// TIA Portal V16 export
// export: Created 2021-08-10T12:25:23.3020932Z, ExportSetting WithDefaults, DisplayName Totally Integrated Automation Portal, DisplayVersion V16 Update 3, DisplayName TIA Portal Version Control Interface, DisplayVersion V16 Update 2, DisplayName TIA Portal Openness, DisplayVersion V16 Update 3, DisplayName STEP 7 Professional, DisplayVersion V16 Update 3, DisplayName STEP 7 Safety, DisplayVersion V16, DisplayName WinCC Professional, DisplayVersion V16 Update 3
FUNCTION "FC61000_DocGenExample" : Void   // FC61000, LAD
TITLE = Documentation - Gen — Example Documentation (full)
{ S7_Optimized_Access := 'TRUE' }
AUTHOR : M_Gledhill
FAMILY : Documentation
NAME : DocGenExample
VERSION : 1.1
// PRACTICAL SERIES AUTOMATION LIBRARY (PAL)   —   COPYRIGHT 2020 – M. GLEDHILL (MIT LICENCE)
//                   ———— ◆ ————
//  FOR DETAILED DOCUMENTATION — SELECT THE BLOCK IN THE PROJECT TREE AND PRESS SHIFT + F1
//  FULL ONLINE DOCUMENTATION IS AVAILABLE AT: https://practicalseries.com/2001-pal/index.html
// stored: AutoNumber false, IsIECCheckEnabled false, SetENOAutomatically false, UDAEnableTagReadback false
   VAR_INPUT
      SYS_SIGNALS : "UT21000_Dy_SysSignals";   // Common system signals — logic and timing signals
   END_VAR
   VAR_TEMP
      revInfo : "UT01000_St_SysRevision";   // Revision information for this block
      licInfo : "UT01001_St_SysLicence";   // Licence information for this block
      wrkReal : Real;   // Working storage (real)
   END_VAR
BEGIN

REGION Network 1: Block description
   // ▀▀▀▀▀▀▀▀▀▀▀▀▀▀▀▀▀▀▀▀▀▀▀▀▀▀▀▀▀▀▀▀▀▀▀▀▀▀▀▀▀▀▀▀
   // 
   // TITLE:    EXAMPLE DOCUMENTATION FOR USE IN COMMENTS
   // 
   // ▄▄▄▄▄▄▄▄▄▄▄▄▄▄▄▄▄▄▄▄▄▄▄▄▄▄▄▄▄▄▄▄▄▄▄▄▄▄▄▄▄▄▄▄
   // 
   // 
   // 
   // This block contains examples of all the typical forms of documentation used within the PAL
   // software. It provides the following:
   // 
   // CONTENTS (BY NETWORK)
   // 
   // NW 1.    Block Contents
   // NW 2.    Current revision and modification history
   // 
   // 
   // EXAMPLES
   // 
   // NW 3.    Example — Block description — Sections 1 to 3
   // NW 4.    Example — Block description — Sections 4 to 11
   // NW 5.    Example — Current revision and modification history
   // NW 6.    Example — Headings, lists and indented text
   // NW 7.    Example — Body text
   // NW 8.    Example — Standard Tables
   // NW 9.    Example — Other tables
   // NW 10.    Example — Equations
   // NW 11.    Example — Figures
   // 
   // 
   // CHARACTER LISTS
   // 
   // NW 12.    Special characters — Hyphens, whitespace and construction lines
   // NW 13.    Special characters — Arrows, box and block characters
   // NW 14.    Special characters — Currency, punctuation and full-width characters
   // NW 15.    Special characters — Greek, indexing characters and Roman numerals
   // NW 16.    Special characters — Mathematical operators (including vulgar fractions)
   // NW 17.    Special characters — Geometrical and ornamental characters
   // NW 18.    Special characters — Common character widths and additional whitespace characters
   // 
   // 
   // SPECIAL NETWORKS
   // 
   // NW 19.    OB1 NETWORK 1 — Project description
   // NW 20.    OB1 NETWORK 2 — Current revision and modification history
   // 
   // TYPICAL NETWORK COMMENTS
   // 
   // NW 21.    Load the system RTC and store in local variable  [typical network comment]
   // NW 22.    ██ STEP 03340 — DECLARATION (RUNNING)    [sequence network comment]
   // NW 23.       STEP 03340 — ACTION (INITIALISE)           [sequence network comment]
   // NW 24.       STEP 03340 — TRANSITION 01                   [sequence network comment]
   // NW 25.   LICENCE AND CONTACT INFORMATION       [final network]
   // 
   //               ━━━   ⬙⬙⬙⬙⬙⬙   ━━━
   // 
   // 
   // 
   // ▄▄▄▄▄▄▄▄▄▄▄▄▄▄▄▄▄▄▄▄▄▄▄▄▄▄▄▄▄▄▄▄▄▄▄▄▄▄▄▄▄▄▄▄
   // 1.     BLOCK TECHNICAL SUMMARY
   // 
   // 
   //  ――――――――――――――――――――――――――――――――――――――――――
   //  NOMENCLATURE & ADDRESSING
   //  ――――――――――――――――――――――――――――――――――――――――――
   //  BLOCK TITLE         Example Documentation for use in Comments
   //  BLOCK FUNCTION GROUP    Documentation
   //  BLOCK ADDRESS       FC 61000
   //  BLOCK SYMBOL        FC61000_DocGenExample
   //  BLOCK USER ID         DocGenExample
   // 
   //  ――――――――――――――――――――――――――――――――――――――――――
   //  BLOCK TYPE & USAGE
   //  ――――――――――――――――――――――――――――――――――――――――――
   //  BLOCK TYPE         Function (FC)
   //  BLOCK NUMBER        61000
   //  LANGUAGE           LAD
   //  OPTIMISED ACCESS     Yes
   //  PAL USAGE TYPE       Standard block
   // 
   //  ――――――――――――――――――――――――――――――――――――――――――
   //  METRICS
   //  ――――――――――――――――――――――――――――――――――――――――――
   //  EXECUTION TIME       24.48 μs¹
   //  LOAD MEMORY       51.63 kB  (52873 bytes)
   //  WORK MEMORY           0.37 kB      (376 bytes)
   //  ――――――――――――――――――――――――――――――――――――――――――
   //                ¹ Measured on: CPU-1515-2PN (order no. 6ES7 512-2AM02-0AB0)
   // 
   //                ━━━   ⬙⬙⬙⬙⬙⬙   ━━━
   // 
   // 
   // 
   // ▄▄▄▄▄▄▄▄▄▄▄▄▄▄▄▄▄▄▄▄▄▄▄▄▄▄▄▄▄▄▄▄▄▄▄▄▄▄▄▄▄▄▄▄
   // 2.     FUNCTIONAL DESCRIPTION
   // 
   // 
   // FC61000 is a documentation module that contains examples of all the common block and 
   // network comments used throughout the PAL software.
   // 
   // All examples are based upon the Style Guide (Doc. No. PS2001-5-2313-011).
   // 
   // FC61000 also contains lists of the characters available within the Siemens TIA font used within
   // all comment sections.
   // 
   //                ━━━   ⬙⬙⬙⬙⬙⬙   ━━━
   // 
   // 
   // 
   // ▄▄▄▄▄▄▄▄▄▄▄▄▄▄▄▄▄▄▄▄▄▄▄▄▄▄▄▄▄▄▄▄▄▄▄▄▄▄▄▄▄▄▄▄
   // 3.     DETAILED BLOCK DESCRIPTION
   // 
   // 
   // The purpose of this block is to provide an easy point of reference for the various documentation 
   // constructs and styles used within the PAL.
   // 
   // The block itself does not contain any executable code, with the exception of the revision and
   // licence networks, all networks are empty. The block itself does nothing, and its execution will
   // have no effect, other than extending the cycle time.
   // 
   //                ━━━   ⬙⬙⬙⬙⬙⬙   ━━━
   // 
   // 
   // 
   // ▄▄▄▄▄▄▄▄▄▄▄▄▄▄▄▄▄▄▄▄▄▄▄▄▄▄▄▄▄▄▄▄▄▄▄▄▄▄▄▄▄▄▄▄
   // 4.     PARAMETERS
   // 
   // 
   // This block has no parameters.
   // 
   //                ━━━   ⬙⬙⬙⬙⬙⬙   ━━━
   // 
   // 
   // 
   // ▄▄▄▄▄▄▄▄▄▄▄▄▄▄▄▄▄▄▄▄▄▄▄▄▄▄▄▄▄▄▄▄▄▄▄▄▄▄▄▄▄▄▄▄
   // 5.     DATA STRUCTURES AND USAGE (AND INSTANCE DATA BLOCKS)
   // 
   // 
   // The block has the following associated data structure:
   // 
   // 
   //  ――――――――――――――――――――――――――――――――――――――――――
   //  DATA STRUCTURE             DESCRIPTION
   //  ――――――――――――――――――――――――――――――――――――――――――
   //  UT01000_St_SysRevision          Revision information for this block    See FC01001
   //  UT01001_St_SysLicence           Licence information for this block  See FC01001
   //  ――――――――――――――――――――――――――――――――――――――――――
   // 
   // 
   //                ━━━   ⬙⬙⬙⬙⬙⬙   ━━━
   // 
   // 
   // 
   // ▄▄▄▄▄▄▄▄▄▄▄▄▄▄▄▄▄▄▄▄▄▄▄▄▄▄▄▄▄▄▄▄▄▄▄▄▄▄▄▄▄▄▄▄
   // 6.     CONSTANTS AND TEMPORARY (LOCAL) DATA
   // 
   // 
   // The following constants and temporary data storage are used:
   // 
   // 
   //  Temporary (local) data
   //  ――――――――――――――――――――――――――――――――――――――――――
   //  SIGNAL NAME          FUNCTION                  TYPE
   //  ――――――――――――――――――――――――――――――――――――――――――
   //  revInfo             Revision information for the block         UT01000
   //  licInfo           Licensing information for the block      UT01001
   //  wrkReal           Working storage (Real)             Real
   //  ――――――――――――――――――――――――――――――――――――――――――
   // 
   // 
   //  Constants data
   //  ――――――――――――――――――――――――――――――――――――――――――
   //  SIGNAL NAME          FUNCTION                  TYPE
   //  ――――――――――――――――――――――――――――――――――――――――――
   //  _FALSE            Temporary internal "False" signal      Bool
   //  ――――――――――――――――――――――――――――――――――――――――――
   // 
   // 
   //                ━━━   ⬙⬙⬙⬙⬙⬙   ━━━
   // 
   //  
   // 
   // ▄▄▄▄▄▄▄▄▄▄▄▄▄▄▄▄▄▄▄▄▄▄▄▄▄▄▄▄▄▄▄▄▄▄▄▄▄▄▄▄▄▄▄▄
   // 7.     BLOCK CALLS
   // 
   // 
   // There are no PAL block calls from within this block.
   // 
   //                ━━━   ⬙⬙⬙⬙⬙⬙   ━━━
   // 
   // 
   // 
   // ▄▄▄▄▄▄▄▄▄▄▄▄▄▄▄▄▄▄▄▄▄▄▄▄▄▄▄▄▄▄▄▄▄▄▄▄▄▄▄▄▄▄▄▄
   // 8.     ASSOCIATED BLOCKS
   // 
   // 
   // This is a stand-alone block and is not associated with any other blocks.
   // 
   //                ━━━   ⬙⬙⬙⬙⬙⬙   ━━━
   // 
   // 
   // 
   // 9.     SYSTEM BLOCK CALLS AND SYSTEM DATA TYPES
   // 
   // There are no system block calls.
   // 
   //                ━━━   ⬙⬙⬙⬙⬙⬙   ━━━
   // 
   // 
   // 
   // ▄▄▄▄▄▄▄▄▄▄▄▄▄▄▄▄▄▄▄▄▄▄▄▄▄▄▄▄▄▄▄▄▄▄▄▄▄▄▄▄▄▄▄▄
   // 10.     SPECIAL PROPERTIES AND REQUIREMENTS
   // 
   // 
   // 
   // ▂▂▂▂▂▂▂▂▂▂▂▂▂▂▂▂▂▂▂▂▂▂▂▂▂▂▂▂▂▂▂▂▂▂▂▂▂▂▂▂▂▂▂▂
   // 10.1   Block optimisation
   // 
   // 
   // Block optimisation is ACTIVE for this block
   // 
   // 
   // 
   // ▂▂▂▂▂▂▂▂▂▂▂▂▂▂▂▂▂▂▂▂▂▂▂▂▂▂▂▂▂▂▂▂▂▂▂▂▂▂▂▂▂▂▂▂
   // 10.2   Calling requirements
   // 
   // 
   // There are no special calling requirements for this block.
   // 
   //                ━━━   ⬙⬙⬙⬙⬙⬙   ━━━
   // 
   // 
   // 
   // ▄▄▄▄▄▄▄▄▄▄▄▄▄▄▄▄▄▄▄▄▄▄▄▄▄▄▄▄▄▄▄▄▄▄▄▄▄▄▄▄▄▄▄▄
   // 11.     EXAMPLE USAGE
   // 
   // 
   // The following shows a typical deployment of FC61000:
   // 
   // 
   //                        ┌────────────
   //    ────────────────────┤ FC61000 
   //                        ├──────────
   //      "DB21001_DY_StdGlobalData".SysSignals ─┤ SYS_SIGNALS
   //                        │
   //                        │               │
   //                        │               │
   //                                     │
   //                        ─────────────┘
   // 
   //               ━━━   ⬙⬙⬙⬙⬙⬙   ━━━
   // 
   // 
   // ██████████████ █ █ █ █  END   █ █ █ █ ██████████████
END_REGION

REGION Network 2: Current revision and modification history
   // ▄▄▄▄▄▄▄▄▄▄▄▄▄▄▄▄▄▄▄▄▄▄▄▄▄▄▄▄▄▄▄▄▄▄▄▄▄▄▄▄▄▄▄▄
   // MODIFICATION HISTORY
   // 
   // The revision data shown here, in the network comments, contains additional information 
   // reflecting the software development workflow under the version control system (VCS) employed 
   // to track all software changes.
   // 
   // The VCS in use is the Git Source Code Management system in conjunction with the GitHub online 
   // hosting system. The software in its entirety is available in the GitHub remote repository:
   // 
   //      https://github.com/practicalseries/PS2001-pal-software
   // 
   // The repository is public and can be freely copied (forked in GitHub terminology) and used 
   // under the MIT licence. 
   // 
   // The MIT licence is reproduced in full in the last network of this software module.
   // 
   // 
   //  ―――――――――――――――――――――――――――――――――――――――――――
   //  DATE       REVISION             MASTER BRANCH     DEV
   //          (nnn.amm)   COMMIT TAG    (Base ---> Merge)    BRANCH   Author
   //  ———————————————————————————————————————————
   //  2021.08.10    001.102   D0008A-000.103   D0008 N/A     D0008A   M. Gledhill
   //                        Constants table added to network 8
   // 
   //  2021.05.18    001.101   D0005A-000.102   D0005 N/A     D0005A   M. Gledhill
   //                        OB1 secondary commit revision added
   //                        OB1 document list updated
   // 
   //  2021.02.18    001.000   D0002      D0001 D0002  None    M. Gledhill
   //                        FC61000 — RELEASED FOR USE
   //                          Block imported form 000.125-Db
   //  ———————————————————————————————————————————
   //   Where: nnn  =  Major revision
   //         a  =  Type (1-7 Development, 8 Proving, 9 Qualification, 0 Release)
   //       mm  =  Minor revision (must be 00 if a = 0)
   //         Block properties version number should be set to nn.a (only one decimal place)
   // 
   // ▄▄▄▄▄▄▄▄▄▄▄▄▄▄▄▄▄▄▄▄▄▄▄▄▄▄▄▄▄▄▄▄▄▄▄▄▄▄▄▄▄▄▄▄
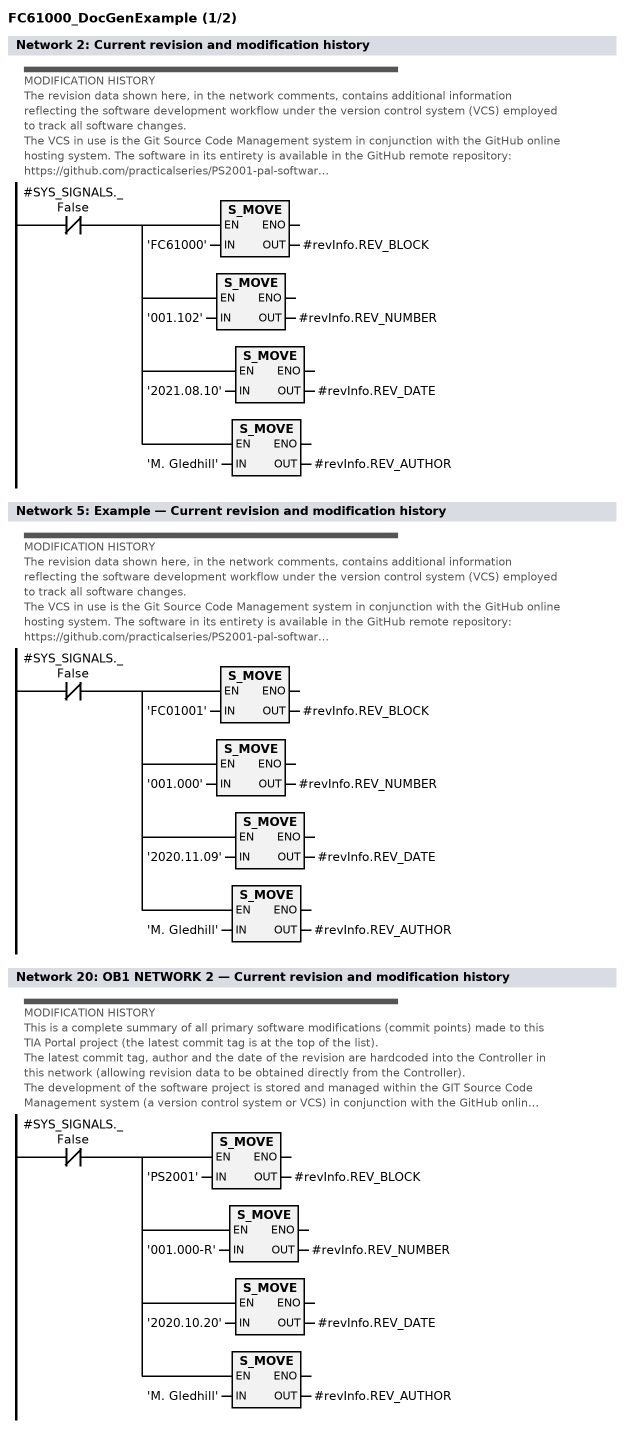
   RUNG wire#powerrail
      I_Contact( #SYS_SIGNALS._False )
      wire#w1
      S_Move(in := 'FC61000', out => #revInfo.REV_BLOCK)
   END_RUNG
   RUNG wire#w1
      S_Move(in := '001.102', out => #revInfo.REV_NUMBER)
   END_RUNG
   RUNG wire#w1
      S_Move(in := '2021.08.10', out => #revInfo.REV_DATE)
   END_RUNG
   RUNG wire#w1
      S_Move(in := 'M. Gledhill', out => #revInfo.REV_AUTHOR)
   END_RUNG
   // the same network as SCL:
   IF NOT #SYS_SIGNALS._False THEN
       #revInfo.REV_BLOCK := 'FC61000';
       #revInfo.REV_NUMBER := '001.102';
       #revInfo.REV_DATE := '2021.08.10';
       #revInfo.REV_AUTHOR := 'M. Gledhill';
   END_IF;
END_REGION

REGION Network 3: Example — Block description — Sections 1 to 3
   // | ▀▀▀▀▀▀▀▀▀▀▀▀▀▀▀▀▀▀▀▀▀▀▀▀▀▀▀▀▀▀▀▀▀▀▀▀▀▀▀▀▀▀▀▀
   // 
   // TITLE:    SUBROUTINE — EVENT TIMER USING RTC
   // 
   // ▄▄▄▄▄▄▄▄▄▄▄▄▄▄▄▄▄▄▄▄▄▄▄▄▄▄▄▄▄▄▄▄▄▄▄▄▄▄▄▄▄▄▄▄
   //  
   // 
   // 
   // This block (FC18151_SubTimeEventRTC) is a subroutine block that times the duration of an event 
   // to nanosecond resolution.
   // 
   // The block records the time the event started (rising edge of the TRIGGER signal), the time the 
   // event ended (falling edge of the TRIGGER signal) and calculates the duration of the event (end 
   // time minus the start time).
   // 
   // The start and end times are read from the real time clock of the controller.
   // 
   // This is a subroutine block.
   // 
   //                ━━━   ⬙⬙⬙⬙⬙⬙   ━━━
   // 
   // 
   // 
   // ▄▄▄▄▄▄▄▄▄▄▄▄▄▄▄▄▄▄▄▄▄▄▄▄▄▄▄▄▄▄▄▄▄▄▄▄▄▄▄▄▄▄▄▄
   // 1.     BLOCK TECHNICAL SUMMARY
   // 
   // 
   //  ――――――――――――――――――――――――――――――――――――――――――
   //  NOMENCLATURE & ADDRESSING
   //  ――――――――――――――――――――――――――――――――――――――――――
   //  BLOCK TITLE         Subroutine Event Timer using RTC
   //  BLOCK FUNCTION GROUP    Subroutine
   //  BLOCK ADDRESS       FC18151
   //  BLOCK SYMBOL        FC18151_SubTimeEventRTC
   //  BLOCK USER ID         SubTimeEventRTC
   // 
   //  ――――――――――――――――――――――――――――――――――――――――――
   //  BLOCK TYPE & USAGE
   //  ――――――――――――――――――――――――――――――――――――――――――
   //  BLOCK TYPE         Function (FC)
   //  BLOCK NUMBER        18151
   //  LANGUAGE           LAD
   //  OPTIMISED ACCESS     Yes
   //  PAL USAGE TYPE       Standard block
   // 
   //  ――――――――――――――――――――――――――――――――――――――――――
   //  METRICS
   //  ――――――――――――――――――――――――――――――――――――――――――
   //  EXECUTION TIME       18.41 μs¹
   //  LOAD MEMORY       23.11 kB  (23667 bytes)
   //  WORK MEMORY           0.43 kB      (442 bytes)
   //  ――――――――――――――――――――――――――――――――――――――――――
   //                ¹ Measured on: CPU-1515-2PN (order no. 6ES7 512-2AM02-0AB0)
   // 
   //                ━━━   ⬙⬙⬙⬙⬙⬙   ━━━
   // 
   // 
   // 
   // ▄▄▄▄▄▄▄▄▄▄▄▄▄▄▄▄▄▄▄▄▄▄▄▄▄▄▄▄▄▄▄▄▄▄▄▄▄▄▄▄▄▄▄▄
   // 2.     FUNCTIONAL DESCRIPTION
   // 
   // 
   // FC18151 is the Subroutine Event Timer using RTC block, it simply records the duration of an event 
   // with a high degree of accuracy. The event being timed is a Boolean signal passed to the block as 
   // the TRIGGER parameter.
   // 
   // Three times are recorded for the event, the start time (rising edge of the TRIGGER parameter), the 
   // end time (falling edge of the TRIGGER parameter) and the duration of the event (end time minus 
   // the start time). The duration is calculated on the falling edge of the TRIGGER parameter, 
   // immediately after the end time is recorded.
   // 
   // The start and end times are read from the Controller’s internal real time clock (RTC) and are 
   // stored in DTL (date time long) format, this format contains year, month, day, hours, minutes, 
   // seconds, milliseconds, microseconds and nano seconds.
   // 
   // The duration is stored in LTime (long time, 64-bit) format, and is very accurate, it resolves to 
   // days, hours, minutes, seconds milliseconds, microseconds and nanoseconds, it keeps this 
   // resolution irrespective of the duration.
   // 
   // The duration is also calculated as a real number in seconds (or fractions thereof); this is a 
   // more convenient format for holding the duration, but is not as accurate as the LTime format.
   // 
   //                ━━━   ⬙⬙⬙⬙⬙⬙   ━━━
   // 
   // 
   // 
   // ▄▄▄▄▄▄▄▄▄▄▄▄▄▄▄▄▄▄▄▄▄▄▄▄▄▄▄▄▄▄▄▄▄▄▄▄▄▄▄▄▄▄▄▄
   // 3.     DETAILED BLOCK DESCRIPTION
   // 
   // 
   // The purpose of this block is to determine with a high degree of accuracy the duration of an event, 
   // the event itself must be in the form of a Boolean trigger signal, the rising edge of the signal is 
   // considered to be the start of the event and the falling edge the end of the event.
   // 
   // The event signal is passed to the block as the TRIGGER parameter. 
   // The block returns five values, these are stored in a UDT passed to the block in the 
   // DYNAMIC_DATA parameter: 
   // 
   // 
   //  ――――――――――――――――――――――――――――――――――――――――――
   //  PARAM         ASSOCIATED UDT            ASSOCIATED DATA BLOCK
   //  ――――――――――――――――――――――――――――――――――――――――――
   //  DYNAMIC_DATA     UT38151_Dy_SubTimeEventRTC       DB38151_Dy_SubTimeEventRTC
   //  ――――――――――――――――――――――――――――――――――――――――――
   // 
   // 
   // The block returns the following data:
   // 
   // 
   //  UT38151_Dy_SubTimeEventRTC
   //  ―――――――――――――――――――――――――――――――――――――――――― 
   //  SIGNAL NAME          FUNCTION                     TYPE
   //  ――――――――――――――――――――――――――――――――――――――――――
   //  status_Running      STATUS — The event timer is running         Bool
   // 
   //  actual_StartTime      ACTUAL — Time at which the TRIGGER signal        DTL
   //                      went high (event start time)
   // 
   //  actual_EndTime        ACTUAL — Time at which the TRIGGER signal     DTL
   //                      went low (event end time)
   // 
   //  actual_Duration        ACTUAL — Event duration              LTime
   // 
   //  actual_DurationSec       ACTUAL — Event duration in seconds           REAL
   //  ――――――――――――――――――――――――――――――――――――――――――
   //  Block returned signals.
   // 
   // 
   // 
   // ▂▂▂▂▂▂▂▂▂▂▂▂▂▂▂▂▂▂▂▂▂▂▂▂▂▂▂▂▂▂▂▂▂▂▂▂▂▂▂▂▂▂▂▂
   // 3.1     Timing an event
   // 
   // 
   // The block constantly monitors the TRIGGER parameter; if a rising edge is seen on the TRIGGER 
   // parameter (point ① in the figure below), the Controller RTC is read and its value is stored in 
   // actual_StartTime, at the same time the running signal (status_Running) is activated.
   // 
   // The block continues to monitor the TRIGGER parameter, when a falling edge is detected 
   // (point ②), the RTC is read once more and its value is stored in actual_EndTime, and the running 
   // signal (status_Running) is deactivated.
   // 
   // Once the end time is stored, the following calculation is carried out:
   // 
   // 
   // ┌───────────────────────────┐
   // │ actual_Duration =  actual_EndTime ─ actual_StartTime    │
   // └───────────────────────────┘
   // 
   // 
   //                     ①            ②
   //   TRIGGER │             ┏━━━━━━━━━━━━┓
   //         │             ┃               ┃
   //         │             ┃               ┃
   //         │             ┃               ┃
   //         │             ┃               ┃                              
   //         ┼━━━━━━━━━━━━╶╶╶╶╶╶╶╶╶╶╶╶╶━━━━━━━━━━ time
   //                  ↗             ↖
   //            actual_StartTime ╎            ╎ actual_EndTime
   //    DTL#2020-04-18-09:34:25.899548353        DTL#2020-04-18-09:34:36.004744916
   // 
   //                    ╎               ╎                      actual_Duration
   //                                      LT#10S_105MS_196US_563NS
   //                    ╎               ╎  
   //                                                     actual_DurationSec
   //                    ╎               ╎                              10.10519
   // 
   //         │status_Running      ┏━━━━━━━━━━━━┓
   //         │             ┃               ┃
   //         │             ┃               ┃
   //         │             ┃               ┃
   //         │             ┃               ┃
   //         ┼━━━━━━━━━━━━╶╶╶╶╶╶╶╶╶╶╶╶╶━━━━━━━━━━
   // 
   // 
   // 
   // ▂▂▂▂▂▂▂▂▂▂▂▂▂▂▂▂▂▂▂▂▂▂▂▂▂▂▂▂▂▂▂▂▂▂▂▂▂▂▂▂▂▂▂▂
   // 3.1     Date and time data types
   // 
   // 
   // Both the start and end times (actual_StartTime and actual_EndTime) are of the type DTL 
   // (date time long), this itself is a data structure in the form:
   // 
   // 
   //  DTL Data Structure
   //  ――――――――――――――――――――――――――――――――――――――――――
   //  SIGNAL NAME          FUNCTION                     TYPE
   //  ――――――――――――――――――――――――――――――――――――――――――
   //  YEAR             Year (returns a value in the range 1970 to 2262)     UInt
   //  MONTH            Month (1-12 representing Jan to Dec)        USInt
   //  DAY              Day of month (1-31)                USInt
   //  WEEKDAY          Day of week (1-7, where 1=Sunday, 7=Saturday)    USInt
   //  HOUR           Hour of day (0-23)                   USInt
   //  MINUTE           Minutes (0-59)                   USInt
   //  SECOND            Seconds (0-59)                  USInt
   //  NANOSECOND        Nanoseconds (0-999,999,999)           UDint
   //  ――――――――――――――――――――――――――――――――――――――――――
   // 
   // 
   // When displayed, it has the format:
   // 
   //       DTL#2020-04-18-09:34:25.899548353
   // 
   //  I.e.      18th April 2020 at 09:43:25 AM and 899,548,353 ns.
   // 
   // The calculated duration (actual_Duration) is of data type LTime (long time).
   // 
   // The LTime data type is essentially an 8-byte number (64-bit number) that stores a time value in 
   // nanoseconds. In the above example, the actual_Duration has the formatted value of:
   // 
   //       LT#10S_105MS_196US_563NS
   // 
   //  I.e.      10 seconds, 105 milliseconds, 196 microseconds and 563 nanoseconds.
   // 
   // It is shown in this format, because TIA portal understands the LTime data type and is able to 
   // interpret the value as days, hours, minute, seconds, milliseconds, microseconds and 
   // nanoseconds. 
   // 
   // In practice, the actual_Duration simply (in this example) holds a very large number:
   // 
   //       10,105,196,563
   // 
   // This is the duration of the event in nanoseconds (i.e. 10,105,196,563 nanoseconds). To convert 
   // the number to seconds, simply divide by 1,000,000,000 (or 1 × 10^9); this would give:
   // 
   //       10.105196563 seconds
   // 
   // The reason the duration is specified as an LTime rather that DTL is that, somewhat confusingly, 
   // DTL is a relative measure of time (relative to 1st January, 1970), if the above duration were 
   // represented as a DTL value it would read:
   // 
   //       DTL#1970-01-01-00:00:10.105196563
   // 
   // Hours, minutes and seconds are OK, but the date part doesn’t make sense (to make it 
   // meaningful, 1970 must be subtracted from the YEAR value and 1 from both the MONTH and 
   // DAY values).
   // 
   // The LTime data type can store a duration of up to 106,751 days (about 300 years) and while not 
   // perfect, it seems long enough for most practical situations (possibly not for geological 
   // applications).
   // 
   // The actual_Duration in LTime format is very accurate, but it is an unwieldly data type, to provide a 
   // more user friendly (although less accurate) format, the actual_Duration signal is converted to a 
   // real number giving the duration in seconds, this is stored in the actual_DurationSec signal. In the 
   // above example: 
   // 
   //       actual_DurationSec has the value 10.10519 seconds
   // 
   // It is less accurate, it does not resolve to nanoseconds; however, it is easier to use and display 
   // and is accurate enough for most applications.
   // 
   // 
   // 
   // ▁▁▁▁▁▁▁▁▁▁▁▁▁▁▁▁▁▁▁▁▁▁▁▁▁▁▁▁▁▁▁▁▁▁▁▁▁▁▁▁▁▁▁▁
   // A note on real numbers
   // 
   // 
   // The LTime format is very accurate, it is basically counting nanoseconds, and because it is 64-bits 
   // long it can count up to very high values (about 584 years at nanosecond resolution).
   // 
   // Real numbers however, are limited to 32-bits and suffer from precision loss, this results from the 
   // fact that the real number has an accuracy of “about” 7 decimal digits, for example 20365.45, 
   // 20.43728, 1.482967, 0.3356428, &c. Essentially, the bigger the number, the fewer the decimal 
   // places — a total of 7 decimal digits.
   // 
   // Very big and very small numbers can be represented by adding trailing zeros for big numbers 
   // (e.g. 3275625000) and leading zeros for small numbers (0.000003275625) in both these 
   // examples, there are only 7 decimal digits, just shifted effectively left or right.
   // 
   // This type of representation is usually handled by applying scientific notation, the number 
   // 1,568,497,000,000 would be represented as 1.568497 × 10^12, it only has 7 decimal digits, 
   // the number 1,568,497,132,792, would be represented as exactly the same value, the 132,792 
   // part of the number cannot be resolved and are lost.
   // 
   //                ━━━   ⬙⬙⬙⬙⬙⬙   ━━━
END_REGION

REGION Network 4: Example — Block description — Sections 4 to 11
   // ▄▄▄▄▄▄▄▄▄▄▄▄▄▄▄▄▄▄▄▄▄▄▄▄▄▄▄▄▄▄▄▄▄▄▄▄▄▄▄▄▄▄▄▄
   // 4.     PARAMETERS
   // 
   // 
   // The following parameters are associated with the block:
   // 
   //  
   //  ――――――――――――――――――――――――――――――――――――――――――
   //  PARAM         FUNCTION                    TYPE      IN-OUT 
   //  ――――――――――――――――――――――――――――――――――――――――――
   //  SYS_SIGNALS      Common system signals              UT21000    In
   //           logic and timing signals for parametric access
   // 
   //  TRIGGER       Event trigger signal (a rising edge marks the     Bool   In
   //           start of the event, the falling edge the end)
   // 
   //  STATIC_DATA     Data structure that holds the configuration data     UT02001    In
   // 
   //  DYNAMIC_DATA      Stores the results of the event timing       UT38151    InOut
   //  ――――――――――――――――――――――――――――――――――――――――――
   // 
   // 
   //                ━━━   ⬙⬙⬙⬙⬙⬙   ━━━
   // 
   // 
   // 
   // ▄▄▄▄▄▄▄▄▄▄▄▄▄▄▄▄▄▄▄▄▄▄▄▄▄▄▄▄▄▄▄▄▄▄▄▄▄▄▄▄▄▄▄▄
   // 5.     DATA STRUCTURES AND USAGE (AND INSTANCE DATA BLOCKS)
   // 
   // 
   // The block has the following associated data structure:
   // 
   // 
   //  ――――――――――――――――――――――――――――――――――――――――――
   //  DATA STRUCTURE             DESCRIPTION
   //  ――――――――――――――――――――――――――――――――――――――――――
   //  UT01000_St_SysRevision          Revision information for this block    See FC01001
   //  UT01001_St_SysLicence           Licence information for this block  See FC01001
   //  UT21000_Dy_SysSignals           System signals for logic and timing  See FC01001
   //  UT38151_Dy_SubTimeEventRTC        Dynamic data structure for the event timing block
   //  ――――――――――――――――――――――――――――――――――――――――――
   // 
   // 
   // 
   // ▂▂▂▂▂▂▂▂▂▂▂▂▂▂▂▂▂▂▂▂▂▂▂▂▂▂▂▂▂▂▂▂▂▂▂▂▂▂▂▂▂▂▂▂
   // 5.1     UT38151_Dy_TimeEventRTC
   // 
   // 
   // Stores the timing values for the event:
   // 
   // 
   //  UT38151_Dy_TimeEventRTC
   //  ――――――――――――――――――――――――――――――――――――――――――
   //  SIGNAL NAME          FUNCTION                     TYPE
   //  ――――――――――――――――――――――――――――――――――――――――――
   //  status_Running      STATUS — The event timer is running         Bool
   // 
   //  actual_StartTime      ACTUAL — Time at which the TRIGGER signal        DTL
   //                      went high (event start time)
   // 
   //  actual_EndTime        ACTUAL — Time at which the TRIGGER signal     DTL
   //                      went low (event end time)
   // 
   //  actual_Duration        ACTUAL — Event duration              LTime
   // 
   //  actual_DurationSec       ACTUAL — Event duration in seconds           REAL
   //  ――――――――――――――――――――――――――――――――――――――――――
   // 
   // 
   //                ━━━   ⬙⬙⬙⬙⬙⬙   ━━━
   // 
   // 
   // 
   // ▄▄▄▄▄▄▄▄▄▄▄▄▄▄▄▄▄▄▄▄▄▄▄▄▄▄▄▄▄▄▄▄▄▄▄▄▄▄▄▄▄▄▄▄
   // 6.     CONSTANTS AND TEMPORARY (LOCAL) DATA
   // 
   // 
   // The following constants and temporary data storage are used:
   // 
   // 
   //  Temporary (local) data
   //  ――――――――――――――――――――――――――――――――――――――――――
   //  SIGNAL NAME          FUNCTION                  TYPE
   //  ――――――――――――――――――――――――――――――――――――――――――
   //  revInfo             Revision information for the block         UT01000
   //  licInfo           Licensing information for the block      UT01001
   //  wrkInt           Working storage area (integer)          Int
   //  wrkReal           Working storage (Real)             Real
   //  wrkLInt            Working storage area (long integer)        LInt
   //  ――――――――――――――――――――――――――――――――――――――――――
   // 
   // 
   //                ━━━   ⬙⬙⬙⬙⬙⬙   ━━━
   // 
   // 
   // 
   // ▄▄▄▄▄▄▄▄▄▄▄▄▄▄▄▄▄▄▄▄▄▄▄▄▄▄▄▄▄▄▄▄▄▄▄▄▄▄▄▄▄▄▄▄
   // 7.     BLOCK CALLS
   // 
   // 
   // There are no PAL block calls from within this block.
   // 
   //                ━━━   ⬙⬙⬙⬙⬙⬙   ━━━
   // 
   // 
   // 
   // ▄▄▄▄▄▄▄▄▄▄▄▄▄▄▄▄▄▄▄▄▄▄▄▄▄▄▄▄▄▄▄▄▄▄▄▄▄▄▄▄▄▄▄▄
   // 8.     ASSOCIATED BLOCKS
   // 
   // 
   // This is a stand-alone block and is not associated with any other blocks.
   // 
   //                ━━━   ⬙⬙⬙⬙⬙⬙   ━━━
   // 
   // 
   // 
   // ▄▄▄▄▄▄▄▄▄▄▄▄▄▄▄▄▄▄▄▄▄▄▄▄▄▄▄▄▄▄▄▄▄▄▄▄▄▄▄▄▄▄▄▄
   // 9.     SYSTEM BLOCK CALLS AND SYSTEM DATA TYPES
   // 
   // 
   // The following calls are made to system blocks:
   // 
   // 
   //  System block calls
   //  ――――――――――――――――――――――――――――――――――――――――――
   //  BLOCK          TITLE             DESCRIPTION  
   //  ――――――――――――――――――――――――――――――――――――――――――
   //  RD_LOC_T             Read the local RTC time    Reads the CPU real time clock 
   //  ――――――――――――――――――――――――――――――――――――――――――
   // 
   // 
   // There are no special system data types used.
   // 
   //                ━━━   ⬙⬙⬙⬙⬙⬙   ━━━
   // 
   // 
   // 
   // ▄▄▄▄▄▄▄▄▄▄▄▄▄▄▄▄▄▄▄▄▄▄▄▄▄▄▄▄▄▄▄▄▄▄▄▄▄▄▄▄▄▄▄▄
   // 10.     SPECIAL PROPERTIES AND REQUIREMENTS
   // 
   // 
   // 
   // ▂▂▂▂▂▂▂▂▂▂▂▂▂▂▂▂▂▂▂▂▂▂▂▂▂▂▂▂▂▂▂▂▂▂▂▂▂▂▂▂▂▂▂▂
   // 10.1   Block optimisation
   // 
   // 
   // Block optimisation is ACTIVE for this block
   // 
   // 
   // 
   // ▂▂▂▂▂▂▂▂▂▂▂▂▂▂▂▂▂▂▂▂▂▂▂▂▂▂▂▂▂▂▂▂▂▂▂▂▂▂▂▂▂▂▂▂
   // 10.2   Calling requirements
   // 
   // 
   // There are no special calling requirements for this block.
   // 
   // 
   // 
   // ▂▂▂▂▂▂▂▂▂▂▂▂▂▂▂▂▂▂▂▂▂▂▂▂▂▂▂▂▂▂▂▂▂▂▂▂▂▂▂▂▂▂▂▂
   // 10.3   Other properties
   // 
   // 
   // This block does not require the usual SYS_SIGNALS logic and timing data.
   // 
   //                ━━━   ⬙⬙⬙⬙⬙⬙   ━━━
   // 
   // 
   // 
   // ▄▄▄▄▄▄▄▄▄▄▄▄▄▄▄▄▄▄▄▄▄▄▄▄▄▄▄▄▄▄▄▄▄▄▄▄▄▄▄▄▄▄▄▄
   // 11.     EXAMPLE USAGE
   // 
   // 
   // The following shows a typical deployment of FC18151:
   // 
   //                      ┌─────────────
   //        ──────────────┤ FC18151
   //                      ├───────────
   //                 %M100.0    │
   //               "Event001"   ─┤ TRIGGER
   //                      │
   //     "DB38151_Dy_TimeEventRTC".Event001 ─┤ DYNAMIC_DATA
   //                      │
   //                      │             │
   //                                    │
   //                           ─────────┘
   // 
   //               ━━━   ⬙⬙⬙⬙⬙⬙   ━━━
   // 
   // 
   // ██████████████ █ █ █ █  END   █ █ █ █ ██████████████
END_REGION

REGION Network 5: Example — Current revision and modification history
   // ▄▄▄▄▄▄▄▄▄▄▄▄▄▄▄▄▄▄▄▄▄▄▄▄▄▄▄▄▄▄▄▄▄▄▄▄▄▄▄▄▄▄▄▄
   // MODIFICATION HISTORY
   // 
   // 
   // The revision data shown here, in the network comments, contains additional information 
   // reflecting the software development workflow under the version control system (VCS) employed 
   // to track all software changes.
   // 
   // The VCS in use is the Git Source Code Management system in conjunction with the GitHub online 
   // hosting system. The software in its entirety is available in the GitHub remote repository:
   // 
   //      https://github.com/practicalseries/PS2001-pal-software
   // 
   // The repository is public and can be freely copied (forked in GitHub terminology) and used 
   // under the MIT licence. 
   // 
   // The MIT licence is reproduced in full in the last network of this software module.
   // 
   // 
   //  ―――――――――――――――――――――――――――――――――――――――――――
   //  DATE       REVISION             MASTER BRANCH     DEV
   //          (nnn.amm)   COMMIT TAG    (Base ---> Merge)    BRANCH   Author
   //  ———————————————————————————————————————————
   //  2020.11.09    001.000   D0003      D0002 D0003  None    M. Gledhill
   //                        FC01001 — RELEASED FOR USE
   //                          Merge back to master branch
   //  
   //  2020.11.09    001.000   D0002A-001.000   D0002 N/A     D0002A   M. Gledhill
   //                        FC01001 — Post test released for use
   // 
   //  2020.11.08    000.801   D0002A-000.801   D0002 N/A     D0002A   M. Gledhill
   //                        FC01001 — Released for SMT
   // 
   //  2020.11.04    000.102   D0002A-000.102   D0002 N/A     D0002A   M. Gledhill
   //                        FC01001 — Incremental build
   // 
   //  2020.11.03    000.101   D0002A-000.101   D0002 N/A     D0002A   M. Gledhill
   //                        FC01001 — Block created
   //  ———————————————————————————————————————————
   //   Where: nnn  =  Major revision
   //         a  =  Type (1-7 Development, 8 Proving, 9 Qualification, 0 Release)
   //       mm  =  Minor revision (must be 00 if a = 0)
   //         Block properties version number should be set to nn.a (only one decimal place)
   // 
   // ▄▄▄▄▄▄▄▄▄▄▄▄▄▄▄▄▄▄▄▄▄▄▄▄▄▄▄▄▄▄▄▄▄▄▄▄▄▄▄▄▄▄▄▄
   RUNG wire#powerrail
      I_Contact( #SYS_SIGNALS._False )
      wire#w1
      S_Move(in := 'FC01001', out => #revInfo.REV_BLOCK)
   END_RUNG
   RUNG wire#w1
      S_Move(in := '001.000', out => #revInfo.REV_NUMBER)
   END_RUNG
   RUNG wire#w1
      S_Move(in := '2020.11.09', out => #revInfo.REV_DATE)
   END_RUNG
   RUNG wire#w1
      S_Move(in := 'M. Gledhill', out => #revInfo.REV_AUTHOR)
   END_RUNG
   // the same network as SCL:
   IF NOT #SYS_SIGNALS._False THEN
       #revInfo.REV_BLOCK := 'FC01001';
       #revInfo.REV_NUMBER := '001.000';
       #revInfo.REV_DATE := '2020.11.09';
       #revInfo.REV_AUTHOR := 'M. Gledhill';
   END_IF;
END_REGION

REGION Network 6: Example — Headings, lists and indented text
   // ▀▀▀▀▀▀▀▀▀▀▀▀▀▀▀▀▀▀▀▀▀▀▀▀▀▀▀▀▀▀▀▀▀▀▀▀▀▀▀▀▀▀▀▀
   // ↳
   // TITLE:    HEADINGS, LISTS AND INDENTED TEXT
   // ↳
   // ▄▄▄▄▄▄▄▄▄▄▄▄▄▄▄▄▄▄▄▄▄▄▄▄▄▄▄▄▄▄▄▄▄▄▄▄▄▄▄▄▄▄▄▄[3 empty lines below]
   // ↳
   // ↳
   // ↳
   // Lorem ipsum dolor sit amet, consectetur adipiscing elit, sed do eiusmod tempor incididunt ut 
   // labore et dolore magna aliqua. Euismod lacinia at quis risus sed. Semper feugiat nibh sed 
   // pulvinar proin gravida hendrerit.
   // ↳
   //                ━━━   ⬙⬙⬙⬙⬙⬙   ━━━[1 empty line above]
   // ↳
   // ↳
   // ↳
   // ▄▄▄▄▄▄▄▄▄▄▄▄▄▄▄▄▄▄▄▄▄▄▄▄▄▄▄▄▄▄▄▄▄▄▄▄▄▄▄▄▄▄▄▄[3 empty lines above, 2 after title]
   // 1.     [MAIN SECTION — ALL UPPERCASE — IF UNNUMBERED STARTS AT LEFT EDGE]
   // 10.     [MAIN SECTION — ALL UPPERCASE — IF UNNUMBERED STARTS AT LEFT EDGE]
   // ↳
   // ↳
   // Lorem ipsum dolor sit amet, consectetur adipiscing elit, sed do eiusmod tempor incididunt ut 
   // labore et dolore magna aliqua. Euismod lacinia at quis risus sed. Semper feugiat nibh sed 
   // pulvinar proin gravida hendrerit.
   // ↳
   //                ━━━   ⬙⬙⬙⬙⬙⬙   ━━━[1 empty line above]
   // ↳
   // ↳
   // ↳
   // ▂▂▂▂▂▂▂▂▂▂▂▂▂▂▂▂▂▂▂▂▂▂▂▂▂▂▂▂▂▂▂▂▂▂▂▂▂▂▂▂▂▂▂▂[3 empty lines above, 2 after title]
   // 1.1     [Subsection, two single digits   — Sentence case — if unnumbered, starts at left edge]
   // 10.1   [Subsection, one double digit   — Sentence case — if unnumbered, starts at left edge]
   // 10.10    [Subsection, two double digits — Sentence case — if unnumbered, starts at left edge]
   // ↳
   // ↳
   // Lorem ipsum dolor sit amet, consectetur adipiscing elit, sed do eiusmod tempor incididunt ut 
   // labore et dolore magna aliqua. Euismod lacinia at quis risus sed. Semper feugiat nibh sed 
   // pulvinar proin gravida hendrerit.
   // ↳
   //                ━━━   ⬙⬙⬙⬙⬙⬙   ━━━[1 empty line above]
   // ↳
   // ↳
   // ↳
   // ▁▁▁▁▁▁▁▁▁▁▁▁▁▁▁▁▁▁▁▁▁▁▁▁▁▁▁▁▁▁▁▁▁▁▁▁▁▁▁▁▁▁▁▁[3 empty lines above, 2 after title]
   // 1.1.1     [Inline, three single digits   — Sentence case — if unnumbered, starts at left edge]
   // 10.1.1   [Inline, one double digit   — Sentence case — if unnumbered, starts at left edge]
   // 10.10.1   [Inline, two double digits    — Sentence case — if unnumbered, starts at left edge]
   // 10.10.10 [Inline, three double digits — Sentence case — if unnumbered, starts at left edge]
   // ↳
   // ↳
   //    •   [Lists — non-numbered]
   //    ① [Lists — numbered]
   //    1.  [Lists — numbered single digit   — less than 10 entries]
   //      1.  [Lists — numbered single digit   — 10 or more entries]
   //    10.  [Lists — numbered double digit — 10 or more entries]
   // 
   //    1.  Communication handling
   //      Executes system to system communications (Controller to Controller, point-to-point,
   //      ProfiBus FMS &c.)
   //    2.  Subroutine functions
   //      Various subroutines (called by other block) to execute particular functions 
   //      (subroutines are organised into similar function areas)
   //    3.  Normal (non-error) interrupt functions
   //      Usually associated with specific OBs, interrupts generated by standard system events
   //      (time of day, cyclic, hardware &c.)
   // 
   // Note:    Bipolar and unipolar instruments have different tolerances, a 0-20 mA unipolar signal
   //      has a full instrument range of 16 mA and the 2.5% tolerance will thus be ±0.4 mA 
   // 
   // ――――――――――
   // ¹         Footnotes can use the characters ¹, ² and ³ to indicate the footnote number
   //      Second lines are identical to those for notes.
   // ――――――――――
   // ↳
   //                ━━━   ⬙⬙⬙⬙⬙⬙   ━━━
   // ↳
   // ↳
   // ██████████████ █ █ █ █  END   █ █ █ █ ██████████████
   // ↳
END_REGION

REGION Network 7: Example — Body text
   // ▀▀▀▀▀▀▀▀▀▀▀▀▀▀▀▀▀▀▀▀▀▀▀▀▀▀▀▀▀▀▀▀▀▀▀▀▀▀▀▀▀▀▀▀
   // 
   // TITLE:    BODY TEXT (AN EXAMPLE)
   // 
   // ▄▄▄▄▄▄▄▄▄▄▄▄▄▄▄▄▄▄▄▄▄▄▄▄▄▄▄▄▄▄▄▄▄▄▄▄▄▄▄▄▄▄▄▄
   // 
   // 
   // Normal (body) text is left justified to the left hand edge of the comment area; manual line-breaks
   // must be inserted when the text exceeds the range of the title bars (lines at the top of this block
   // and above each section and subsection — exactly 44 em-spaces).
   // 
   // The following fragment highlights this: 
   // 
   // The alignments in Figure 7.4 are such that the leading edge (left side) of any indented character
   // is aligned with the leading edge of an em-space in a line of em-spaces that span the page (this
   // can be seen with the chequered patterns in the screen shot — all indents line up with the left
   // edge of an em-space).
   // 
   // The problem with this is that the alphanumeric characters are not all the same width and
   // generally, they are not one em-space wide (there are no characters that are one em wide, not
   // even the M, which is odd given that that is how the em unit was derived, see here).
   // With the TIA Portal font, one em is exactly the same width as four normal space characters (a 
   // normal space being the character entered when the space bar is pressed). The alphanumeric 
   // characters (and in fact, all the characters) in the TIA Portal font have the peculiarity that they are
   // all a multiple of ⅓ of a normal space , the “i" for example is one normal space wide, “a” is 2⅓
   // normal space characters wide and “m” is 2⅔ normal space characters wide.
   // 
   // This “feature?” of the font is a distinct advantage; it means that is possible to always bring things
   // back into true alignment by using the range of whitespace characters. There are five such 
   // whitespace characters.
   // 
   // The width of the page is approximately 3.38 lowercase alphabets:
   // 
   // abcdefghijklmnopqrstuvwxyzabcdefghijklmnopqrstuvwxyzabcdefghijklmnopqrstuvwxyzabcdefghij
   // 
   // This averages at about 78 (non-space) characters per line.
   // 
   // A comment field can contain 65000 characters (approx.) including spaces and line breaks.
   // 
   // This broadly equates to 670 lines of standard text, approximately 13000 words.
   // ↳
   //                ━━━   ⬙⬙⬙⬙⬙⬙   ━━━
   // ↳
   // ↳
   // ██████████████ █ █ █ █  END   █ █ █ █ ██████████████
   // ↳
END_REGION

REGION Network 8: Example — Standard Tables
   // ▀▀▀▀▀▀▀▀▀▀▀▀▀▀▀▀▀▀▀▀▀▀▀▀▀▀▀▀▀▀▀▀▀▀▀▀▀▀▀▀▀▀▀▀
   // 
   // TITLE:    STANDARD TABLES (EXAMPLES)
   // 
   // ▄▄▄▄▄▄▄▄▄▄▄▄▄▄▄▄▄▄▄▄▄▄▄▄▄▄▄▄▄▄▄▄▄▄▄▄▄▄▄▄▄▄▄▄
   // 
   // 
   // 
   // Tables always have 2 blank lines above and 2 blank lines below.
   // 
   // ▌▌▌▌▌▌▌▌▌▌▌▌▌▌▌▌▌▌PARAMETER TABLE▐▐▐▐▐▐▐▐▐▐▐▐▐▐▐▐▐▐
   // ↳
   // ↳
   //  ――――――――――――――――――――――――――――――――――――――――――
   //  PARAM         FUNCTION                    TYPE      IN-OUT 
   //  ――――――――――――――――――――――――――――――――――――――――――
   //  SYS_SIGNALS      The system logic and timing signals for       UT21000    In
   //           parametric access
   // 
   //  RAW_ANALOG      The unscaled analogue input (input word         Word     In
   //           address for the IO card to which the instrument 
   //           is connected)
   // 
   //  RAW_MIN     Minimum value of the analogue input range      Int      In
   //           (see Table 3.1 to Table 3.3 for typical values)
   // 
   //  RAW_MAX       Maximum value of the analogue input range      Int      In
   //           (see Table 3.1 to Table 3.3 for typical values)
   // 
   //  SCALE_MIN    Calibrated lower value of the instrument       Real      In
   //           range in engineering units
   // 
   //  SCALE_MAX      Calibrated upper value of the instrument      Real      In
   //           range in engineering units
   // 
   //  STATIC_DATA     The static data associated with the PID loop       UT10001 In
   // 
   //  DYNAMIC_DATA      Stores the results of the event timing       UT38151    InOut
   //  ――――――――――――――――――――――――――――――――――――――――――
   // ↳
   // ↳
   // 
   // ▌▌▌▌▌▌▌▌▌▌▌▌▌▌▌▌▌ DATA STRUCTURE LIST ▐▐▐▐▐▐▐▐▐▐▐▐▐▐▐▐▐
   // ↳
   // ↳
   //  ――――――――――――――――――――――――――――――――――――――――――
   //  DATA STRUCTURE             DESCRIPTION
   //  ――――――――――――――――――――――――――――――――――――――――――
   //  UT01000_St_SysRevision          Revision information for this block    See FC01000
   //  UT01001_St_SysLicence           Licence information for this block  See FC01000
   //  UT21000_Dy_SysSignals           System signals for logic and timing  See FC01000
   // 
   //  UT02001_St_InstAnalogRead      Static data structure for an analogue instrument.
   //                     Holds configuration information, instrument ranges 
   //                     and scaling, alarm/warning thresholds &c.
   // 
   //  UT22001_Dy_InstAnalogRead        Dynamic data structure for an analogue instrument.
   //                     Current scaled instrument reading, alarm status, 
   //                     operating modes, timer values &c.
   //  ――――――――――――――――――――――――――――――――――――――――――
   // ↳
   // ↳
   // 
   // ▌▌▌▌▌▌▌▌▌▌   DATA STRUCTURE CONTENTS AND INSTANCE DBs   ▐▐▐▐▐▐▐▐▐▐
   // ↳
   // ↳
   //  UT38151_Dy_TimeEventRTC
   //  ――――――――――――――――――――――――――――――――――――――――――
   //  SIGNAL NAME          FUNCTION                     TYPE
   //  ――――――――――――――――――――――――――――――――――――――――――
   //  status_Running      STATUS — The event timer is running         Bool
   // 
   //  actual_StartTime      ACTUAL — Time at which the TRIGGER signal        DTL
   //                      went high (event start time)
   // 
   //  actual_EndTime        ACTUAL — Time at which the TRIGGER signal     DTL
   //                      went low (event end time)
   // 
   //  actual_Duration        ACTUAL — Event duration              LTime
   // 
   //  actual_DurationSec       ACTUAL — Event duration in seconds           REAL
   //  ――――――――――――――――――――――――――――――――――――――――――
   // ↳
   // ↳
   // 
   // ▌▌▌▌▌▌▌▌▌▌▌▌▌▌▌  CONSTANTS AND LOCAL DATA  ▐▐▐▐▐▐▐▐▐▐▐▐▐▐▐
   // 
   // [Keep local and constant data function description to one line and no gaps between rows]
   // ↳
   // ↳
   //  CONSTANTS DATA
   //  ――――――――――――――――――――――――――――――――――――――――――
   //  SIGNAL NAME       Value    FUNCTION                  TYPE
   //  ――――――――――――――――――――――――――――――――――――――――――
   //  k_TIME_OP_MIN      0.21      Minimum value for the operation timer     Real
   //  ――――――――――――――――――――――――――――――――――――――――――
   // ↳
   // ↳
   //  TEMPORARY (LOCAL) DATA
   //  ――――――――――――――――――――――――――――――――――――――――――
   //  SIGNAL NAME          FUNCTION                     TYPE
   //  ――――――――――――――――――――――――――――――――――――――――――
   //  wrkPercentPV          Process Variable as a percentage of inst. range     Real
   //  wrkPercentSP          Setpoint as a percentage of PV instrument range     Real
   //  wrkPercentDB         Deadband as a percentage of PV instrument range    Real
   //  wrkGain          Gain (adjusted for reverse/normal Acting)      Real
   //  wrkCycTime          Cyclic execution time (TIME format)         Time
   //  ――――――――――――――――――――――――――――――――――――――――――
   // ↳
   // ↳
   // 
   // ▌▌▌▌▌▌▌▌▌▌▌▌▌▌▌▌▌▌▌  BLOCK LIST  ▐▐▐▐▐▐▐▐▐▐▐▐▐▐▐▐▐▐▐
   // ↳
   // ↳
   //  BLOCK CALLS
   //  ――――――――――――――――――――――――――――――――――――――――――
   //  BLOCK          TITLE             DESCRIPTION  
   //  ――――――――――――――――――――――――――――――――――――――――――
   //  FC18001         StdSubScaleAI        Scales an analogue input signal 
   //                            Continuation line
   //  ――――――――――――――――――――――――――――――――――――――――――
   // ↳
   // ↳
   //  ASSOCIATED BLOCKS
   //  ――――――――――――――――――――――――――――――――――――――――――
   //  BLOCK          TITLE             DESCRIPTION  
   //  ――――――――――――――――――――――――――――――――――――――――――
   //  FC17102         StdCommsWrite65K       Write data partner block
   //                            Continuation line 
   //  ――――――――――――――――――――――――――――――――――――――――――
   // ↳
   // ↳
   // 
   // ▌▌▌▌▌▌▌▌▌▌▌▌▌▌▌▌▌  SYSTEM BLOCK LIST   ▐▐▐▐▐▐▐▐▐▐▐▐▐▐▐▐▐
   // ↳
   // ↳
   //  SYSTEM BLOCK CALLS
   //  ――――――――――――――――――――――――――――――――――――――――――
   //  BLOCK          TITLE             DESCRIPTION  
   //  ――――――――――――――――――――――――――――――――――――――――――
   //  RD_LOC_T             Read the local RTC time    Reads the CPU real time clock 
   //  (FC804)                        Continuation line 
   //                            Continuation line
   //  ――――――――――――――――――――――――――――――――――――――――――
   // ↳
   // ↳
   // 
   // ▌▌▌▌▌▌▌▌▌▌▌▌▌▌▌▌▌▌▌▌▌▌▐▐▐▐▐▐▐▐▐▐▐▐▐▐▐▐▐▐▐▐▐▐
   // ↳
   //                ━━━   ⬙⬙⬙⬙⬙⬙   ━━━
   // ↳
   // ↳
   // ██████████████ █ █ █ █  END   █ █ █ █ ██████████████
   // ↳
END_REGION

REGION Network 9: Example — Other tables
   // ▀▀▀▀▀▀▀▀▀▀▀▀▀▀▀▀▀▀▀▀▀▀▀▀▀▀▀▀▀▀▀▀▀▀▀▀▀▀▀▀▀▀▀▀
   // 
   // TITLE:    OTHER TABLES (EXAMPLES)
   // 
   // ▄▄▄▄▄▄▄▄▄▄▄▄▄▄▄▄▄▄▄▄▄▄▄▄▄▄▄▄▄▄▄▄▄▄▄▄▄▄▄▄▄▄▄▄
   // 
   // 
   // 
   // Tables always have 2 blank lines above and 2 blank lines below.
   // 
   // 
   // ▌▌▌▌▌▌▌▌▌▌▌▌▌▌▌▌▌  TWO COLUMN TABLE ▐▐▐▐▐▐▐▐▐▐▐▐▐▐▐▐▐
   // ↳
   // ↳
   //  ――――――――――――――――――――――――――――――――――――――――――
   //  IO TYPE            DESCRIPTION
   //  ――――――――――――――――――――――――――――――――――――――――――
   //  ET200MP         Standard IO high density IO for the S7-1500 range
   // 
   //  ET200M           Standard IO high density IO for the S7-300 range, 
   //               can be used as remote IO for the S7-1500
   //  ――――――――――――――――――――――――――――――――――――――――――
   // ↳
   // ↳
   // 
   // ▌▌▌▌▌▌▌▌▌▌▌▌▌▌▌▌▌THREE COLUMN TABLE ▐▐▐▐▐▐▐▐▐▐▐▐▐▐▐▐▐
   // 
   // [Numerical table with number alignment to the right]
   // ↳
   // ↳
   //  ――――――――――――――――――――――――――――――――――――――――――
   //  PRESSURE           RAW SIGNAL           SCALED VAL
   //  ――――――――――――――――――――――――――――――――――――――――――
   //  -250.0 Pa                   0             -250.0 Pa
   //        0.0 Pa                  13824            0.0 Pa
   //   250.0 Pa                  27648              250.0 Pa
   //  ――――――――――――――――――――――――――――――――――――――――――
   // ↳
   // ↳
   // 
   // ▌▌▌▌▌▌▌▌▌▌▌▌▌▌▌▌▌ FOUR COLUMN TABLE ▐▐▐▐▐▐▐▐▐▐▐▐▐▐▐▐▐
   // 
   // [Numerical table with number alignment to the right]
   // ↳
   // ↳
   //  ――――――――――――――――――――――――――――――――――――――――――
   //  RAW MIN       RAW MAX      SCALED MIN       SCALED MAX
   //  ――――――――――――――――――――――――――――――――――――――――――
   //        0        27648        -250.0 Pa        250.0 Pa
   //  ――――――――――――――――――――――――――――――――――――――――――
   // ↳
   // ↳
   // 
   // ▌▌▌▌▌▌▌▌▌▌▌▌▌▌▌▌▌  TABLE WITH HEADING  ▐▐▐▐▐▐▐▐▐▐▐▐▐▐▐▐▐
   // 
   // [Numerical table with number alignment to the right]
   // ↳
   // ↳
   //  CURRENT SIGNALS
   //  ――――――――――――――――――――――――――――――――――――――――――
   //  SIGNAL TYPE     SIG MIN VAL      RAW_MIN     SIG MAX VAL     RAW_MAX
   //  ――――――――――――――――――――――――――――――――――――――――――
   //    4-20 mA      4 mA          0          20 mA       27648
   //    0-20 mA      0 mA          0          20 mA       27648
   //  -20 to 20 mA      -20 mA      -27648          20 mA       27648
   //  ――――――――――――――――――――――――――――――――――――――――――
   // ↳
   // ↳
   // 
   // ▌▌▌▌▌▌▌▌▌▌▌▌▌▌▌▌▌▌▌▌▌▌▐▐▐▐▐▐▐▐▐▐▐▐▐▐▐▐▐▐▐▐▐▐
   // ↳
   //                ━━━   ⬙⬙⬙⬙⬙⬙   ━━━
   // ↳
   // ↳
   // ██████████████ █ █ █ █  END   █ █ █ █ ██████████████
   // ↳
END_REGION

REGION Network 10: Example — Equations
   // ▀▀▀▀▀▀▀▀▀▀▀▀▀▀▀▀▀▀▀▀▀▀▀▀▀▀▀▀▀▀▀▀▀▀▀▀▀▀▀▀▀▀▀▀
   // 
   // TITLE:    EQUATIONS (EXAMPLES)
   // 
   // ▄▄▄▄▄▄▄▄▄▄▄▄▄▄▄▄▄▄▄▄▄▄▄▄▄▄▄▄▄▄▄▄▄▄▄▄▄▄▄▄▄▄▄▄
   // 
   // 
   // 
   // ┌─────────────────────────────────────┐
   // │                                                                                                              100                         │
   // │ SigPercent = (Signal ─ PV_RANGE_MIN) ╳ ---------------------------------------------------------------    │
   // │                    (PV_RANGE_MAX ─ PV_RANGE_MIN)    │
   // └─────────────────────────────────────┘
   // 
   // 
   // ┌───────────────────────┐
   // │        2.5               │
   // │ CalcValOOR = ------------ ╳ (RAW_MAX ─ RAW_MIN)   │
   // │       100               │
   // └───────────────────────┘
   // 
   // Mathematical operators:
   //    Large:  ┼ ─ ╳
   //    Small: + − × ÷ ± ≤ ≥
   // ↳
   //                ━━━   ⬙⬙⬙⬙⬙⬙   ━━━
   // ↳
   // ↳
   // ██████████████ █ █ █ █  END   █ █ █ █ ██████████████
   // ↳
END_REGION

REGION Network 11: Example — Figures
   // ▀▀▀▀▀▀▀▀▀▀▀▀▀▀▀▀▀▀▀▀▀▀▀▀▀▀▀▀▀▀▀▀▀▀▀▀▀▀▀▀▀▀▀▀
   // 
   // TITLE:    FIGURES (EXAMPLES)
   // 
   // ▄▄▄▄▄▄▄▄▄▄▄▄▄▄▄▄▄▄▄▄▄▄▄▄▄▄▄▄▄▄▄▄▄▄▄▄▄▄▄▄▄▄▄▄
   // 
   // 
   // 
   // Some example figures, always pad gaps with an EM-SPACE, where text is used add normal 
   // spaces with either a THREE-PER-EM space or a SIX-PER-EM space — one of these will give an
   // exact alignment.
   // 
   // These figures are included to show what is possible.
   // 
   // 
   // Figures have 1 blank line above and 1 below.
   // 
   //   → ┌────────┐
   // ┌───┤   IDLE   │
   // │   └───┬────┘
   // │       ↓
   // │       START
   // │       │
   // │   ┌───┴────┐ →
   // │   │  STARTING     ├───┐
   // │   └───┬────┘   │
   // │       ↓        │
   // │         Run*       ├────────────────────┐
   // │       │        │                    │
   // │   ┌───┴────┐ → │                    │
   // │   │        ├───┴───  Hold  ───┐          │
   // │   │        │             ↓          ↓
   // │   │        │         ┌───┴────┐ ┌───┴────┐
   // │   │        │         │  HOLDING    │ │ ErrHOLDING   │
   // │   │        │         └───┬────┘ └───┬────┘
   // │   │        │             Held*        ErrHeld*
   // │   │        │         ┌───┴────┐ ┌───┴────┐
   // │   │        │         │   HELD    │ │  ErrHELD   │
   // │   │  RUNNING     │         └───┬────┘ └───┬────┘
   // │   │        │              Resume         ErrResume
   // │   │        │         ┌───┴────┐ ┌───┴────┐
   // │  ┌┤        │         │   RESUMING    │ │  ErrRESUMING   │ 
   // │  ││        │         └───┬────┘ └───┬────┘  
   // │  ││        │             │          │
   // │  ││        │ ←           ↓          ↓
   // │  ││        │─────────────┴──────────┘
   // │  │└───┬────┘   Returns to previous step (running or starting)
   // │  ↓    ↓
   // │  │    │
   // │ Complete Complete*     Note: *indicates that the command is issued
   // │  │    │           automatically by the sequence (it
   // │  │┌───┴────┐      can also be triggered manually):
   // │  └┤ COMPLETING  │          1. Run
   // │   └───┬────┘          2. Complete
   // │       ↓               3. Completed
   // ↑     Completed*              4. Held
   // │       │               5. ErrHeld
   // │   ┌───┴────┐          6. Stopped
   // │   │  COMPLETED   │          7. Aborted
   // │   └───┬────┘
   // │       │
   // │              RetIdle*
   // │   ←   ↓
   // ├───────┘
   // │   
   // │
   // │     ABORT ROUTE                  STOPPING ROUTE
   // │Can be triggered in all states except       Can be triggered in all states except
   // │ IDLE, COMPLETED, ABORTING or            IDLE, COMPLETED, ABORTING, 
   // │       ABORTED                 ABORTED, STOPPING or STOPPED
   // │       │                       │
   // │       ↓                       ↓
   // │                Abort                                                                                       Stop
   // │       │                       │
   // │   ┌───┴────┐              ┌───┴────┐
   // ↑   │ ABORTING    │              │  STOPPING    │
   // │   └───┬────┘              └───┬────┘
   // │       ↓                       ↓
   // │              Aborted*                                                                                Stopped*
   // │       │                       │
   // │   ┌───┴────┐              ┌───┴────┐
   // │   │ ABORTED      │              │ STOPPED   │
   // │   └───┬────┘              └───┬────┘
   // │       │                       │
   // │      RetIdle (*)                                                                               RetIdle (*)
   // │  ←    ↓                       ↓
   // └───────┴───────────────────────┘
   // 
   // 
   // 
   // ▌▌▌▌▌▌▌▌▌▌▌▌▌▌▌▌▌▌   INLINE FIGURES ▐▐▐▐▐▐▐▐▐▐▐▐▐▐▐▐▐▐
   // 
   // 
   // 
   // ▂▂▂▂▂▂▂▂▂▂▂▂▂▂▂▂▂▂▂▂▂▂▂▂▂▂▂▂▂▂▂▂▂▂▂▂▂▂▂▂▂▂▂▂
   // 1.1     Step operation and phases
   // 
   // 
   //  ┌─────┐  The sequence progresses from one step to the next if the
   //  │Step n        │  transition logic for the step is TRUE. 
   //  └┬────┘                                                                 
   //   │       In this example, STEP n is active and will remain active
   //         --- T n        until its associated transition (T n) becomes TRUE; at this
   //   │       point the sequence will advance to the next step (STEP n+1)
   //  ┌┴────┐  and execute the actions required of this step. The sequence
   //  │Step n+1    │  will remain in this step until its transition condition is
   //  └┬────┘  true, at which point the sequence will advance again.
   //   │                                                                      
   //         --- T n+1      Each step has a step number, this is an integer value in
   //   │       the range 0 to 29999; step numbers are assigned in specific
   //           Ranges for different operating states of the sequence (IDLE,
   //           STARTING, RUNNING &c.).
   // 
   // Within an individual step, the step has three distinct phases and actions can 
   // be attached to any of these phases (externally to the block). The phases are:
   // 
   // INITIALISING (Phs_INIT)                   ┌──────┐
   // This is activated for a single OB1 scan when the step   │INITIALISING   │
   // is first processed (I.e. on the rising edge of the step     └┬─────┘
   // becoming active).                     │      
   //                           ┌┴─────┐ 
   // PROCESSING (Phs_PROC)               │PROCESSING │
   // This is the main phase of the step, it is activated        └┬─────┘
   // immediately following the INITIALISING phase and remains  │       
   // active until the step TRANSITION condition is TRUE. The     --- T n   
   // PROCESSING phase becomes inactive on the rising edge   │     
   // of the TRANSITION condition.              ┌┴─────┐
   //                           │TERMINATING │    
   // TERMINATING (Phs_TERM)               └──────┘    
   // The TERMINATING phase is activated on the rising edge of the TRANSITION
   // condition (the same condition that terminates the PROCESSING phase). The
   // terminating phase is active for a single OB1 scan.
   // 
   // 
   // [ALTERNATIVE]
   //  ┌──────┐ INITIALISING (Phs_INIT)
   //  │INITIALISING   │ This is activated for a single OB1 scan when the step
   //  └┬─────┘ is first processed (I.e. on the rising edge of the step
   //   │       becoming active).
   //  ┌┴─────┐    
   //  │PROCESSING │ PROCESSING (Phs_PROC)
   //  └┬─────┘ This is the main phase of the step, it is activated 
   //   │       immediately following the INITIALISING phase and remains
   //          --- T n       active until the step TRANSITION condition is TRUE. The
   //   │       PROCESSING phase becomes inactive on the rising edge
   //  ┌┴─────┐ of the TRANSITION condition.
   //  │TERMINATING │    
   //  └──────┘
   // 
   // TERMINATING (Phs_TERM)
   // The TERMINATING phase is activated on the rising edge of the TRANSITION
   // condition (the same condition that terminates the PROCESSING phase). The
   // terminating phase is active for a single OB1 scan.
   // 
   // 
   // 
   // 
   // ▌▌▌▌▌▌▌▌▌▌▌▌▌▌▌▌▌   GRAPHICAL FIGURE   ▐▐▐▐▐▐▐▐▐▐▐▐▐▐▐▐▐
   // 
   //     No. of scans from start of STEP 1
   //     1      2      3     4      5     6       7      8      9
   //   ┼─┼─┼─┼─┼─┼─┼─┼─┼─┼─┼─┼  ─ ─ ┐
   //                                │
   //   ┌─┐                          │
   //   │ │               Phs_INIT
   //  ─┘ └────────────────────                   
   //   ┼─┼─┼─┼─┼─┼─┼─┼─┼─┼─┼─┼                   
   //  
   //     ┌───┐                       S
   //     │   │           Phs_PROC      T
   //  ───┘   └────────────────       E
   //   ┼─┼─┼─┼─┼─┼─┼─┼─┼─┼─┼─┼       P
   //  
   //         ┌─┐                     1
   //         │ │         TRANSITION
   //  ───────┘ └──────────────
   //   ┼─┼─┼─┼─┼─┼─┼─┼─┼─┼─┼─┼
   // 
   //         ┌─┐
   //         │ │         Phs_TERM      │
   //  ───────┘ └──────────────      │
   //   ┼─┼─┼─┼─┼─┼─┼─┼─┼─┼─┼─┼  ─ ─ ┘
   // 
   // 
   //     1      2      3     4      5     6       7      8      9
   //   ┼─┼─┼─┼─┼─┼─┼─┼─┼─┼─┼─┼  ─ ─ ┐
   //                                │
   //           ┌─┐                  │
   //           │ │       Phs_INIT
   //   ────────┘ └────────────                   
   //   ┼─┼─┼─┼─┼─┼─┼─┼─┼─┼─┼─┼                   
   // 
   //             ┌───┐               S
   //             │   │   Phs_PROC      T
   //  ───────────┘   └────────       E
   //   ┼─┼─┼─┼─┼─┼─┼─┼─┼─┼─┼─┼       P
   //                           
   //                 ┌─┐             2
   //                 │ │ TRANSITION
   //  ───────────────┘ └──────      
   //   ┼─┼─┼─┼─┼─┼─┼─┼─┼─┼─┼─┼
   // 
   //                 ┌─┐
   //                 │ │ Phs_TERM      │
   //  ───────────────┘ └──────      │
   //   ┼─┼─┼─┼─┼─┼─┼─┼─┼─┼─┼─┼  ─ ─ ┘
   // 
   // 
   // 
   // ▌▌▌▌▌▌▌▌▌▌▌▌▌▌▌▌▌▌    PAL LOGO    ▐▐▐▐▐▐▐▐▐▐▐▐▐▐▐▐▐▐
   // 
   //          ⠀⠀⠀⠀⠀⠀⠀⠀⠀⠀⠀⠀⠀⠀⠀⠀⠀⠀⠀⠀⠀⠀⠀⠀⠀⠀⠀⠀⠀⣀⣀⣀
   //       ⠀⠀⠀⠀⠀⠀⠀⠀⠀⠀⠀⠀⠀⠀⠀⠀⠀⠀⠀⠀⠀⠀⠀⠀⠀⠀⠀⣤⣶⣿⣿⣿⣿⣿⣿⣤
   //       ⠀⠀⠀⠀⠀⠀⠀⠀⠀⠀⠀⠀⠀⠀⠀⠀⠀⠀⠀⠀⠀⠀⠀⠀⠀⠀⣶⣿⣿⣿⣿⣿⣿⣿⣿⣿⣶
   //       ⠀⠀⠀⠀⠀⠀⠀⠀⠀⠀⠀⠀⠀⠀⠀⠀⠀⠀⠀⠀⠀⠀⠀⠀⠀⠀⣿⣿⣿⣿⣿⣿⣿⣿⣿⣿⣿
   //       ⠀⠀⠀⠀⠀⠀⠀⠀⠀⠀⠀⠀⠀⠀⠀⠀⠀⠀⠀⠀⠀⠀⠀⠀⠀⣀⠛⣿⣿⣿⣿⣿⣿⣿⣿⣿⠿
   //       ⠀⠀⠀⠀⠀⠀⠀⠀⠀⠀⠀⠀⠀⠀⠀⠀⠀⠀⠀⠀⠀⠀⣀⣶⣿⣿⣤⠉⠿⣿⣿⣿⣿⣿⠿⠛⣤⣶
   //       ⠀⠀⠀⠀⠀⠀⠀⠀⠀⠀⠀⠀⠀⠀⠀⠀⠀⠀⠀⠀⣤⣿⣿⣿⣿⣿⣿⣿⣶⣤⠉⠉⠉⠀⠤⣿⣿⣿⣿⣶⣀⣀⣀⣀⣀⣀⣀⣀
   //       ⠀⠀⠀⠀⠀⠀⠀⠀⠀⠀⠀⠀⠀⠀⠀⠀⠀⣀⣶⣿⣿⣿⣿⣿⣿⣿⣿⣿⣿⠉⠀⠀⠀⠀⠀⠉⠿⣿⣿⣿⣿⣿⣿⣿⣿⣿⣿⣿⣶
   //       ⠀⠀⠀⠀⠀⠀⠀⠀⠀⠀⠀⠀⠀⠀⠀⠀⠛⠿⣿⣿⣿⣿⣿⣿⣿⣿⣿⠿⠀⠀⠀⠀⠀⠀⠀⠀⠀⣿⣿⣿⣿⣿⣿⣿⣿⠿⠿⣿⣿⣤
   //       ⠀⠀⠀⠀⠀⠀⠀⠀⠀⣀⣤⣶⣿⣿⣿⣿⣶⣶⣤⠉⠿⣿⣿⣿⣿⣿⠛⠀⠀⠀⠀⠀⠀⠀⠀⠀⠀⣿⣿⣿⣿⠉⠀⠀⠀⠀⠀⠉⣿⣿⣤
   //       ⠀⠀⠀⠀⠀⠀⠀⣀⣶⣿⣿⣿⣿⣿⣿⣿⣿⣿⣿⣿⣤⠉⣿⣿⣿⠛⠀⠀⠀⠀⠀⠀⠀⠀⠀⠀⣿⣿⣿⣿⣿⠀⠀⠀⠀⠀⠀⠀⠀⠿⠿
   //       ⠀⠀⠀⠀⠀⠀⣀⣿⣿⣿⣿⣿⣿⣿⣿⣿⣿⣿⣿⣿⣿⣿⠀⣿⠉⠀⠀⠀⠀⠀⠀⠀⠀⠀⠀⠀⣿⣿⣿⣿⣿
   //       ⠀⠀⠀⠀⠀⠀⣿⣿⣿⣿⣿⣿⣿⣿⣿⣿⣿⣿⣿⣿⣿⣿⣀⠀⠀⠀⠀⠀⠀⠀⠀⠀⠀⠀⠀⠀⠉⠛⠿⣿⣿⣿⣤
   //       ⠀⠀⠀⠀⠀⠀⣿⣿⣿⣿⣿⣿⣿⣿⣿⣿⣿⣿⣿⣿⣿⣿⠿⠀⠀⠀⠀⠀⠀⠀⠀⠀⠀⠀⠀⠀⠀⠀⠀⠀⠉⠛⠿⣿
   //       ⠀⠀⠀⠀⠀⠀⠛⣿⣿⣿⣿⣿⣿⣿⣿⣿⣿⣿⣿⣿⣿⣿
   //       ⠀⠀⠀⠀⠀⠀⠀⠛⣿⣿⣿⣿⣿⣿⣿⣿⣿⣿⣿⣿⠿⠉
   //       ⠀⠀⠀⠀⠀⠀⠀⠀⠀⠛⠿⣿⣿⣿⣿⣿⣿⣿⠿⠉
   //       ⠀⠀⠀⠀⠀⠀⠀⠀⠀⠀⠀⣀⣉⣉⣉⣉⣉⣀
   //       ⠀⠀⠀⠀⠀⠀⠀⠀⠀⣤⣿⣿⣿⣿⣿⣿⣿⣿⣀⠛⣿⣿⣿⣿⣿⣿⣿⣿⣿⣿⣿⣿⣿⣿⣿⣿⣿⣿⣿⣿⣿⣿⣿⣿⣿⣿⣿⣿⣿⣶⣤⣀⠀⠀⠀⠀
   //       ⠀⠀⠀⠀⠀⠀⠀⠀⣤⣿⣿⣿⠿⠉⠉⣿⣿⣿⣿⣤⠉⠿⠿⠿⠿⠿⠿⠿⠿⠿⠿⠿⠿⠿⠿⠿⠿⠿⠿⠿⠿⠿⠿⠿⠿⠿⠿⣿⣿⣿⣿⣿⣿⣀⠀⠀
   //       ⠀⠀⠀⠀⠀⠀⠀⣶⣿⣿⣿⠛⠀⠀   ⠀⠀⠿⣿⣿⣿⣤⠀⠀⠀⠀⠀⠀⣶⣶⣶⣶⣤⠀⠀⠀⠀ ⣶⣶⣶         ⣶⣶⠀⠀⠀⠀⠀⠿⣿⣿⣿⣿⣶⠀
   //       ⠀⠀⠀⠀⠀⠀⣿⣿⣿⣿⠛⠀⠀⠀⠀   ⠀⠀⠛⣿⣿⣿⣶⠀⠀⠀⠀⠀⣿⣿⣿⠿⣿⣿⠀⠀⣤⣿⣿⣿⣤       ⣿⣿⠀⠀⠀⠀⠀⠀ ⠿⣿⣿⣿⣿⣤
   //       ⠀⠀⠀⠀⠀⣿⣿⣿⣿⠉⠀⠀⠀⠀⠀   ⠀⠀⠀⠛⣿⣿⣿⣿⠀⠀⠀⠀⣿⣿⣿⣶⣿⣿⠀⠀⣿⣿⠉⣿⣿       ⣿⣿⠀⠀⠀⠀⠀     ⣿⣿⣿⣿⣿
   //       ⠀⠀⠀⣀⣿⣿⣿⣿⠉⠀⠀⠀⠀⠀⠀⠀⠀   ⠀⠀⠉⣿⣿⣿⣿      ⣿⣿⣿⠛⠛⠀⠀⣶⣿⣿⣿⣿⣿⣶    ⣿⣿⣤⣤⣤      ⣶⣿⣿⣿⣿⠛
   //       ⠀⠀⣤⣿⣿⣿⣿⠉⠀⠀⠀⠀⠀⠀⠀⠀⠀⠀⠀   ⠀⠉⣿⣿⣿⣿⣀ ⠿⠿⠿⠀⠀⠀   ⠿⠿⠉⠉⠉⠿⠿    ⠿⠿⠿⠿⠿ ⠀⣶⣿⣿⣿⣿⠿⠀
   //       ⠀⣤⣿⣿⣿⣿⣿⣶⣤⣤⣤⣤⣤⣤⣤⣤⣤⣤⣤⣤⣶⣿⣿⣿⣿⣿⣀⠀⣶⣶⣶⣶⣶⣶⣶⣶⣶⣶⣶⣶⣶⣶⣶⣶⣶⣶⣶⣶⣿⣿⣿⣿⠉⠀⠀
   //       ⠀⣿⣿⣿⣿⣿⣿⣿⣿⣿⣿⣿⣿⣿⣿⣿⣿⣿⣿⣿⣿⣿⣿⣿⣿⣿⣿⠀⠉⣿⣿⣿⣿⣿⣿⣿⣿⣿⣿⣿⣿⣿⣿⣿⣿⣿⣿⣿⣿⠿⠛⠉⠀⠀⠀⠀
   //       ⠀⠉⠛⠛⠛⠛⠛⠛⠛⠛⠛⠛⠛⠛⠛⠛⠛⠛⠛⠛⠛⠛⠛⠛⠛⠛⠉⠀⠀⠉⠉⠉⠉⠉⠉⠉⠉⠉⠉⠉⠉⠉⠉⠉⠉⠉⠉⠉⠀⠀⠀⠀⠀⠀⠀⠀
   // ↳
   //                ━━━   ⬙⬙⬙⬙⬙⬙   ━━━
   // ↳
   // ↳
   // ██████████████ █ █ █ █  END   █ █ █ █ ██████████████
   // ↳
END_REGION

REGION Network 12: Special characters — Hyphens, whitespace and construction lines
   // ▀▀▀▀▀▀▀▀▀▀▀▀▀▀▀▀▀▀▀▀▀▀▀▀▀▀▀▀▀▀▀▀▀▀▀▀▀▀▀▀▀▀▀▀
   // 
   // TITLE:    SPECIAL CHARACTERS
   // 
   // ▄▄▄▄▄▄▄▄▄▄▄▄▄▄▄▄▄▄▄▄▄▄▄▄▄▄▄▄▄▄▄▄▄▄▄▄▄▄▄▄▄▄▄▄
   // 
   // 
   // The TIA Portal Basic font contains many different types of characters:
   // 
   //    •   Hyphens and whitespace characters
   //    •   Construction lines (these are specially ordered characters, useful for building tables &c.)
   //    •   Arrows
   //    •   Box characters (for drawing box and line diagrams)
   //    •   Block characters
   //    •   Currency
   //    •   Punctuation (extended list)
   //    •   Non-proportional letters and numbers
   //    •   Greek characters
   //    •   Indexing characters
   //    •   Roman numerals
   //    •   Mathematical characters
   //    •   Geometric characters
   //    •   Dingbat characters
   // 
   // The following sections contain a list of these characters for use in TIA Portal comment fields.
   // 
   // Note:    The following tables of characters break the rules for comment fields by exceeding
   //      the prescribed comment field width of 44 em-spaces. This is done to give the 
   //      characters in a more concise form whilst maintaining reasonable descriptions for
   //      the characters
   // 
   // 
   // 
   // ▄▄▄▄▄▄▄▄▄▄▄▄▄▄▄▄▄▄▄▄▄▄▄▄▄▄▄▄▄▄▄▄▄▄▄▄▄▄▄▄▄▄▄▄
   // HYPHENS AND WHITESPACE CHARACTERS
   // 
   // 
   // — Em Dash               █ █ Em Space
   // –   En Dash              █ █   En Space
   // ‐    Hyphen               █ █    Three-Per-Em Space
   // ¬   Soft Hyphen             █ █    Normal Space
   //                       █ █     Six-Per-Em Space
   // 
   // 
   // 
   // ▄▄▄▄▄▄▄▄▄▄▄▄▄▄▄▄▄▄▄▄▄▄▄▄▄▄▄▄▄▄▄▄▄▄▄▄▄▄▄▄▄▄▄▄
   // CONSTRUCTION LINES AND USEFUL LINES
   // 
   // 
   // [Copyable whitespace]
   //  █ █ █ █ █ Em En ThreePerEm SixPerEM
   // [Em-space construction line]
   // ▀▄▀▄▀▄▀▄▀▄▀▄▀▄▀▄▀▄▀▄▀▄▀▄▀▄▀▄▀▄▀▄▀▄▀▄▀▄▀▄▀▄▀▄
   // [Central header — used for examples]
   // ▌▌▌▌▌▌▌▌▌▌▌▌▌▌▌▌▌▌▌▌▌▌▐▐▐▐▐▐▐▐▐▐▐▐▐▐▐▐▐▐▐▐▐▐
   // [Title start]
   // ▀▀▀▀▀▀▀▀▀▀▀▀▀▀▀▀▀▀▀▀▀▀▀▀▀▀▀▀▀▀▀▀▀▀▀▀▀▀▀▀▀▀▀▀
   // [Title end/section over-line]
   // ▄▄▄▄▄▄▄▄▄▄▄▄▄▄▄▄▄▄▄▄▄▄▄▄▄▄▄▄▄▄▄▄▄▄▄▄▄▄▄▄▄▄▄▄
   // [Subsection over-line]
   // ▂▂▂▂▂▂▂▂▂▂▂▂▂▂▂▂▂▂▂▂▂▂▂▂▂▂▂▂▂▂▂▂▂▂▂▂▂▂▂▂▂▂▂▂
   // [Inline section over-line]
   // ▁▁▁▁▁▁▁▁▁▁▁▁▁▁▁▁▁▁▁▁▁▁▁▁▁▁▁▁▁▁▁▁▁▁▁▁▁▁▁▁▁▁▁▁
   // [Table row line]
   //  ――――――――――――――――――――――――――――――――――――――――――
   // [Revision row line]
   //  ―――――――――――――――――――――――――――――――――――――――――――
   // [Flourish divider]
   //                ━━━   ⬙⬙⬙⬙⬙⬙   ━━━
   // [End line]
   // ██████████████ █ █ █ █  END   █ █ █ █ ██████████████
END_REGION

REGION Network 13: Special characters — Arrows, box and block characters
   // ▄▄▄▄▄▄▄▄▄▄▄▄▄▄▄▄▄▄▄▄▄▄▄▄▄▄▄▄▄▄▄▄▄▄▄▄▄▄▄▄▄▄▄▄
   // ARROWS
   // 
   // 
   // ← Left Arrow              ⇐ Left dbl Arrow             ↩ Left Arrow Hook
   // ↑ Up Arrow               ⇑ Up dbl Arrow               ↪ Right Arrow Hook
   // → Right Arrow              ⇒ Right dbl Arrow           ⤣ North West Arrow Hook
   // ↓ Down Arrow             ⇓ Down dbl Arrow             ⤤ North East Arrow Hook
   // ↔ Left Right Arrow             ⇔ Left Right dbl Arrow          ⤥ South East Arrow Hook
   // ↕ Up Down Arrow          ⇕ Up Down dbl Arrow          ⤦ South West Arrow Hook
   // ↖ North West Arrow          ⇖ North West dbl Arrow         ↰    Up Arrow Tip Left
   // ↗ North East Arrow          ⇗ North East dbl Arrow          ↱    Up Arrow Tip Right
   // ↘ South East Arrow          ⇘ South East dbl Arrow         ↲    Down Arrow Tip Left
   // ↙ South West Arrow         ⇙    South West dbl Arrow        ↳ Down Arrow Tip Right
   // ⤡ North West & South East Arrow    ⤂ Left dbl Arrow vert Stroke       ↴ Right Arrow Corner down
   // ⤢ North East & South West Arrow    ⤃ Right dbl Arrow vert Stroke     ↵ Down Arrow Corner Left
   // ⇄ Right Arrow Over Left Arrow       ⤆ Left dbl Arrow From Bar        ↶ Anticlockwise Top Semicircle Arrow
   // ⇅ Up Arrow Left Of down Arrow        ⤇ Right dbl Arrow From Bar         ↷ Clockwise Top Semicircle Arrow
   // ⇆ Left Arrow Over Right Arrow       ⤄ Left Right dbl Arrow vert Stroke    ↺ Anticlockwise Open Circle Arrow
   // ⇇ Left Paired Arrows           ↼ Left Harpoon Barb up         ↻ Clockwise Open Circle Arrow
   // ⇈ Up Paired Arrows             ↽ Left Harpoon Barb down         ⟲ Anticlockwise Gapped Circle Arrow
   // ⇉ Right Paired Arrows         ↾ Up Harpoon Barb Right         ⟳ Clockwise Gapped Circle Arrow
   // ⇊ Down Paired Arrows           ↿ Up Harpoon Barb Left
   // ↤ Left Arrow From Bar           ⇀ Right Harpoon Barb up         ▲  Black Up Triangle 
   // ↥ Up Arrow From Bar          ⇁ Right Harpoon Barb down       ▼  Black Down Triangle
   // ↦ Right Arrow From Bar         ⇂ Down Harpoon Barb Right      ▶  Black Right Triangle
   // ↧ down Arrow From Bar        ⇃ Down Harpoon Barb Left         ◀  Black Left Triangle
   // ↨ Up Down Arrow Base         ⇋ Left Harpoon Over Right Harpoon
   // ↞ Left Two head Arrow          ⇌ Right Harpoon Over Left Harpoon
   // ↟ up Two head Arrow         ↯ Down Zigzag Arrow
   // ↠ Right Two head Arrow
   // ↡ Down Two head Arrow
   // ⤙ Left Arrow-Tail
   // ⤚ Right Arrow-Tail
   // ⤛ Left dbl Arrow-Tail    
   // ⤜ Right dbl Arrow-Tail    
   // ⤝ Left Arrow To Black Diamond    
   // ⤞ Right Arrow To Black Diamond    
   // 
   // ⟵  Long Left Arrow             ↢ Left Arrow Tail             ⌃   Up Arrowhead
   // ⟶  Long Right Arrow          ↣ Right Arrow Tail             ⌄   Down Arrowhead
   // ⟷  Long Left Right Arrow         ⤟ Left Arrow Bar To Black Diamond   ⌅   Projective
   // ⟸  Long Left dbl Arrow         ⤠ Right Arrow Bar To Black Diamond    ⌆   Perspective
   // ⟹  Long Right dbl Arrow          ⤌    Left dbl Dash Arrow         ⟰ Up Quadruple Arrow
   // ⟺  Long Left Right dbl Arrow        ⤍    Right dbl Dash Arrow         ⟱ Down Quadruple Arrow
   // ⟻  Long Left Arrow From Bar       ⤎    Left Triple Dash Arrow        ⤊ Up Triple Arrow
   // ⟼  Long Right Arrow From Bar        ⤏    Right Triple Dash Arrow         ⤋ Down Triple Arrow
   // ⟽  Long Left dbl Arrow From Bar       ⤈    Down Arrow horiz Stroke          ⤈   Down Arrow horiz Stroke
   // ⟾  Long Right dbl Arrow From Bar    ⤉    Up Arrow horiz Stroke             ⤉   Up Arrow horiz Stroke
   // 
   // 
   // 
   // ▄▄▄▄▄▄▄▄▄▄▄▄▄▄▄▄▄▄▄▄▄▄▄▄▄▄▄▄▄▄▄▄▄▄▄▄▄▄▄▄▄▄▄▄
   // BOX CHARACTERS
   // 
   // 
   // ─ Box Light horiz            ╌ Box Light dbl Dash horiz       ⋮     Vert Ellipsis
   // │ Box Light vert             ╎ Box Light dbl Dash vert        ⋯    Midline horiz Ellipsis
   // ╱ Box Light diag top Right Left      ╍ Box Heavy dbl Dash horiz       ⋰     Up Right diag Ellipsis
   // ╲ Box Light diag top Left To btm Right    ╏ Box Heavy dbl Dash vert          ⋱    Down Right diag Ellipsis
   // ╳ Box Light diag Cross          ┄ Box Light Triple Dash horiz      ╴ Box Light Left
   // ━ Box Heavy horiz             ┆ Box Light Triple Dash vert       ╵ Box Light Up
   // ┃ Box Heavy vert           ┅ Box Heavy Triple Dash horiz       ╶ Box Light Right
   // ═ Box dbl horiz               ┇ Box Heavy Triple Dash vert        ╷ Box Light Down
   // ║ Box dbl vert              ┈ Box Light Quadruple Dash horiz     ╸ Box Heavy Left
   //                       ┊ Box Light Quadruple Dash vert       ╹ Box Heavy Up
   //                       ┉ Box Heavy Quadruple Dash horiz      ╺ Box Heavy Right
   //                       ┋ Box Heavy Quadruple Dash vert     ╻ Box Heavy Down
   // 
   // ┌ Box Light Down & Right        ├ Box Light vert & Right         ─ Box Light horiz
   // └ Box Light Up & Right           ┤ Box Light vert & Left        │ Box Light vert
   // ┐ Box Light Down & Left           ┬ Box Light Down & horiz         ┼ Box Light vert & horiz
   // ┘ Box Light Up & Left          ┴ Box Light Up & horiz  
   // ┏ Box Heavy Down & Right         ┣ Box Heavy vert & Right          ━ Box Heavy horiz
   // ┗ Box Heavy Up & Right         ┫ Box Heavy vert & Left         ┃ Box Heavy vert
   // ┓ Box Heavy Down & Left         ┳ Box Heavy Down & horiz       ╋ Box Heavy vert & horiz
   // ┛ Box Heavy Up & Left        ┻ Box Heavy Up & horiz  
   //     
   // ┍ Box Down Light & Right Heavy     ┝ Box vert Light & Right Heavy      ━ Box Heavy horiz
   // ┕ Box Up Light & Right Heavy        ┥ Box vert Light & Left Heavy     │ Box Light vert
   // ┑ Box Down Light & Left Heavy     ┯ Box Down Light & horiz Heavy      ┿ Box vert Light & horiz Heavy
   // ┙ Box Up Light & Left Heavy       ┷ Box Up Light & horiz Heavy  
   // 
   // ┎ Box Down Heavy & Right Light     ┠ Box vert Heavy & Right Light      ─ Box Light horiz
   // ┖ Box Up Heavy & Right Light        ┨ Box vert Heavy & Left Light     ┃ Box Heavy vert
   // ┒ Box Down Heavy & Left Light     ┰ Box Down Heavy & horiz Light      ╂ Box vert Heavy & horiz Light
   // ┚ Box Up Heavy & Left Light       ┸ Box Up Heavy & horiz Light  
   // 
   // ┦ Box Up Heavy & Left Down Light     ┪ Box Up Light & Left Down Heavy     ╀ Box Up Heavy & Down horiz Light
   // ┶ Box Right Heavy & Left Up Light   ┹ Box Right Light & Left Up Heavy   ┾ Box Right Heavy & Left vert Light
   // ┟ Box Down Heavy & Right Up Light     ┡ Box Down Light & Right Up Heavy     ╁ Box Down Heavy & Up horiz Light
   // ┭ Box Left Heavy & Right Down Light    ┲ Box Left Light & Right Down Heavy    ┽ Box Left Heavy & Right vert Light
   //  
   // ┞ Box Up Heavy & Right Down Light     ┢ Box Up Light & Right Down Heavy     ╈ Box Up Light & Down horiz Heavy
   // ┮ Box Right Heavy & Left Down Light    ┱ Box Right Light & Left Down Heavy    ╉ Box Right Light & Left vert Heavy
   // ┧ Box Down Heavy & Left Up Light     ┩ Box Down Light & Left Up Heavy     ╇ Box Down Light & Up horiz Heavy
   // ┵ Box Left Heavy & Right Up Light      ┺ Box Left Light & Right Up Heavy   ╊ Box Left Light & Right vert Heavy
   // 
   // ╼ Box Light Left & Heavy Right                            ╄ Box Right Up Heavy & Left Down Light
   // ╽ Box Light Up & Heavy Down                            ╆ Box Right Down Heavy & Left Up Light
   // ╾ Box Heavy Left & Light Right                            ╅ Box Left Down Heavy & Right Up Light
   // ╿ Box Heavy Up & Light Down                            ╃ Box Left Up Heavy & Right Down Light
   // 
   // ╔ Box dbl Down & Right         ╠ Box dbl vert & Right         ═ Box dbl horiz
   // ╚ Box dbl Up & Right           ╣ Box dbl vert & Left           ║ Box dbl vert
   // ╗ Box dbl Down & Left        ╦ Box dbl Down & horiz         ╬ Box dbl vert & horiz
   // ╝ Box dbl Up & Left          ╩ Box dbl Up & horiz  
   //  
   // ╒ Box Down Single & Right dbl     ╞ Box vert Single & Right dbl      ═ Box dbl horiz
   // ╘ Box Up Single & Right dbl        ╡ Box vert Single & Left dbl        │ Box Light vert
   // ╕ Box Down Single & Left dbl        ╤ Box Down Single & horiz dbl      ╪ Box vert Single & horiz dbl
   // ╛ Box Up Single & Left dbl       ╧ Box Up Single & horiz dbl  
   // 
   // ╓ Box Down dbl & Right Single     ╟ Box vert dbl & Right Single      ─ Box Light horiz
   // ╙ Box Up dbl & Right Single        ╢ Box vert dbl & Left Single        ║ Box dbl vert
   // ╖ Box Down dbl & Left Single        ╥ Box Down dbl & horiz Single      ╫ Box vert dbl & horiz Single
   // ╜ Box Up dbl & Left Single       ╨ Box Up dbl & horiz Single  
   // 
   // 
   // 
   // ▄▄▄▄▄▄▄▄▄▄▄▄▄▄▄▄▄▄▄▄▄▄▄▄▄▄▄▄▄▄▄▄▄▄▄▄▄▄▄▄▄▄▄▄
   // BLOCK CHARACTERS
   // 
   // 
   // ▀ Top Half Block             ❘    Light vert Bar              ❘ ❘     En Space
   // ▄ Btm Half Block            ❙    Medium vert Bar           ❘ ❘   Em Space
   // ▐ Right Half Block          ❚   Heavy vert Bar  
   // ▌ Left Half Block    
   // 
   // ▔ Top One Eighth Block        ▉ Left Seven Eighths Block
   // ▁ Btm One Eighth Block          ▊ Left Three Quarters Block
   // ▂ Btm One Quarter Block        ▋ Left Five Eighths Block
   // ▃ Btm Three Eighths Block      ▌ Left Half Block
   // ▄ Btm Half Block            ▍ Left Three Eighths Block
   // ▅ Btm Five Eighths Block         ▎ Left One Quarter Block
   // ▆ Btm Three Quarters Block       ▏ Left One Eighth Block
   // ▇ Btm Seven Eighths Block        ▕ Right One Eighth Block
   // █ Full Block
   // ░ Light Shade
   // ▒ Medium Shade    
   // ▓ Dark Shade    
   // 
   // 
   // ██████████████ █ █ █ █  END   █ █ █ █ ██████████████
END_REGION

REGION Network 14: Special characters — Currency, punctuation and full-width characters
   // ▄▄▄▄▄▄▄▄▄▄▄▄▄▄▄▄▄▄▄▄▄▄▄▄▄▄▄▄▄▄▄▄▄▄▄▄▄▄▄▄▄▄▄▄
   // CURRENCY
   // 
   // 
   // ₳   Austral Sign             €   Euro Sign              ₦  Naira Sign
   // ₵   Cedi Sign               ₠  Euro-Currency Sign          ₪  New Shekel Sign
   // ¢   Cent Sign              ₣  French Franc Sign           ₧   Peseta Sign
   // ₡   Colon Sign               ₰   German Penny Sign           ₱   Peso Sign
   // ₢   Cruzeiro Sign           ₲   Guarani Sign              £  Pound Sign
   // ¤  Currency Sign             ₴   Hryvnia Sign            ₨    Rupee Sign
   // $   Dollar Sign            ₭   Kip Sign              ₮   Tugrik Sign
   // ₫   Dong Sign             ₤   Lira Sign             ₩  Won Sign
   // ₯ Drachma Sign            ₥  Mill Sign              ¥   Yen Sign
   // 
   // 
   // 
   // ▄▄▄▄▄▄▄▄▄▄▄▄▄▄▄▄▄▄▄▄▄▄▄▄▄▄▄▄▄▄▄▄▄▄▄▄▄▄▄▄▄▄▄▄
   // PUNCTUATION AND COMMON SYMBOLS
   // 
   // 
   // #  Hash Sign             "   Quote                 §   Section Sign
   // $   Dollar Sign            “    Left dbl quote             ¶   Pilcrow Sign
   // %  Percent Sign            ”    Right dbl quote
   // &   Ampersand             '    Apostrophe  
   // *   Asterisk              ‘    Left Single quote          †   Dagger
   // ~   Tilde                 ’    Right Single quote           ‡   Dbl Dagger
   // +   Plus Sign               ‹    Single Left Angle quote       •   Bullet
   // -    Hyphen/minus            ›    Single Right Angle quote        ·    Middle Dot
   // =   Equals Sign                                ‣   Triangular Bullet
   // <   Less-Than Sign           ´   Acute Accent              ⁃    Hyphen Bullet
   // >   Greater-Than Sign           `   Grave Accent
   // (    Left Parenthesis
   // )    Right Parenthesis            ©  Copyright Sign           ⁎   Low Asterisk
   // [    Left Square Bracket           ®  Registered Sign  
   // ]    Right Square Bracket         ℀  Account Of               ․    One Dot Leader
   // {   Left Curly Bracket          ℁  Addressed To The Subject      ‥   Two Dot Leader
   // }   Right Curly Bracket          ℂ  Dbl-Struck Capital C           …  Horiz Ellipsis
   // 〈    Left Angle Bracket           ℄   Centre Line Symbol  
   // 〉    Right Angle Bracket            ℅  Care Of               ※  Reference Mark
   // ⁅    Left Square Bracket Quill        ℗  Sound Recording Copyright       ‼   Dbl Exclamation Mark
   // ⁆    Right Square Bracket Quill      ™  Trade Mark Sign            ‽   Interrobang
   // ,    Comma                                 ⁇  Dbl Question Mark
   // .    Full Stop                                   ⁈   Question Exclamation Mark
   // :    Colon                                  ⁉  Exclamation Question Mark
   // ;    Semicolon    
   // !    Exclamation Mark            ⁑   Two Asterisks Aligned vertically     |    Vert Line
   // ?   Question Mark           ⁂   Asterism               ¦    Broken Bar
   // @  Commercial At                              ‖    Dbl vert Line
   // ^   Circumflex Accent            ⁀  Character Tie              ‗   Dbl Low Line
   // /    Solidus               ‿  Undertie             ⁞    Vert Four Dots
   // \    Reverse Solidus            ⁐  Close Up
   // _   Underscore
   // ― Horiz Bar    
   // ¯   Macron
   // ‾   Overline
   // 
   // 
   // 
   // ▄▄▄▄▄▄▄▄▄▄▄▄▄▄▄▄▄▄▄▄▄▄▄▄▄▄▄▄▄▄▄▄▄▄▄▄▄▄▄▄▄▄▄▄
   // NON-PROPORTIONAL (FULL-WIDTH) LETTERS
   // 
   // 
   // Ａ Fullwidth Capital Letter A        ａ Fullwidth Small Letter A       ＂ Fullwidth quote
   // Ｂ Fullwidth Capital Letter B        ｂ Fullwidth Small Letter B       ＇ Fullwidth Apostrophe
   // Ｃ Fullwidth Capital Letter C        ｃ Fullwidth Small Letter C       ＃ Fullwidth Number Sign
   // Ｄ Fullwidth Capital Letter D       ｄ Fullwidth Small Letter D       ＄ Fullwidth Dollar Sign
   // Ｅ Fullwidth Capital Letter E        ｅ Fullwidth Small Letter E       ％ Fullwidth Percent Sign
   // Ｆ Fullwidth Capital Letter F        ｆ Fullwidth Small Letter F       ＆ Fullwidth Ampers&
   // Ｇ Fullwidth Capital Letter G       ｇ Fullwidth Small Letter G       ＊ Fullwidth Asterisk
   // Ｈ Fullwidth Capital Letter H       ｈ Fullwidth Small Letter H          ～ Fullwidth Tilde
   // Ｉ Fullwidth Capital Letter I         ｉ Fullwidth Small Letter I        ＋ Fullwidth Plus Sign
   // Ｊ Fullwidth Capital Letter J         ｊ Fullwidth Small Letter J        － Fullwidth Hyphen-Minus
   // Ｋ Fullwidth Capital Letter K        ｋ Fullwidth Small Letter K       ＝ Fullwidth Equals Sign
   // Ｌ Fullwidth Capital Letter L        ｌ Fullwidth Small Letter L       ＜ Fullwidth Less-Than Sign
   // Ｍ Fullwidth Capital Letter M       ｍ Fullwidth Small Letter M         ＞ Fullwidth Greater-Than Sign
   // Ｎ Fullwidth Capital Letter N       ｎ Fullwidth Small Letter N          （ Fullwidth Left Parenthesis
   // Ｏ Fullwidth Capital Letter O       ｏ Fullwidth Small Letter O       ） Fullwidth Right Parenthesis
   // Ｐ Fullwidth Capital Letter P        ｐ Fullwidth Small Letter P       ［ Fullwidth Left Square Bracket
   // Ｑ Fullwidth Capital Letter Q       ｑ Fullwidth Small Letter Q         ］ Fullwidth Right Square Bracket
   // Ｒ Fullwidth Capital Letter R        ｒ Fullwidth Small Letter R       ｛ Fullwidth Left Curly Bracket
   // Ｓ Fullwidth Capital Letter S        ｓ Fullwidth Small Letter S       ｝ Fullwidth Right Curly Bracket
   // Ｔ Fullwidth Capital Letter T        ｔ Fullwidth Small Letter T        ， Fullwidth Comma
   // Ｕ Fullwidth Capital Letter U       ｕ Fullwidth Small Letter U       ． Fullwidth Full Stop
   // Ｖ Fullwidth Capital Letter V        ｖ Fullwidth Small Letter V       ： Fullwidth Colon
   // Ｗ Fullwidth Capital Letter W       ｗ Fullwidth Small Letter W         ； Fullwidth Semicolon
   // Ｘ Fullwidth Capital Letter X        ｘ Fullwidth Small Letter X       ！ Fullwidth Exclamation Mark
   // Ｙ Fullwidth Capital Letter Y        ｙ Fullwidth Small Letter Y       ？ Fullwidth Question Mark
   // Ｚ Fullwidth Capital Letter Z        ｚ Fullwidth Small Letter Z       ＠ Fullwidth Commercial At
   //                                         ＾ Fullwidth Circumflex Accent
   // ０ Fullwidth Digit Zero         ５ Fullwidth Digit Five          ／ Fullwidth Solidus
   // １ Fullwidth Digit One         ６ Fullwidth Digit Six         ＼ Fullwidth Reverse Solidus
   // ２ Fullwidth Digit Two          ７ Fullwidth Digit Seven         ＿ Fullwidth Low Line
   // ３ Fullwidth Digit Three          ８ Fullwidth Digit Eight           ｜ Fullwidth vert Line
   // ４ Fullwidth Digit Four         ９ Fullwidth Digit Nine         ❘ ❘   Fullwidth space    
   // 
   // 
   // ██████████████ █ █ █ █  END   █ █ █ █ ██████████████
END_REGION

REGION Network 15: Special characters — Greek, indexing characters and Roman numerals
   // ▄▄▄▄▄▄▄▄▄▄▄▄▄▄▄▄▄▄▄▄▄▄▄▄▄▄▄▄▄▄▄▄▄▄▄▄▄▄▄▄▄▄▄▄
   // GREEK CHARACTERS
   // 
   // 
   // Α  Greek Capital Letter Alpha        α   Greek Small Letter Alpha
   // Β   Greek Capital Letter Beta       β   Greek Small Letter Beta
   // Γ   Greek Capital Letter Gamma       γ   Greek Small Letter Gamma
   // Δ  Greek Capital Letter Delta      δ   Greek Small Letter Delta
   // Ε   Greek Capital Letter Epsilon     ε   Greek Small Letter Epsilon
   // Ζ   Greek Capital Letter Zeta       ζ   Greek Small Letter Zeta
   // Η  Greek Capital Letter Eta       η   Greek Small Letter Eta
   // Θ  Greek Capital Letter Theta      θ   Greek Small Letter Theta
   // Ι    Greek Capital Letter Iota         ι    Greek Small Letter Iota
   // Κ   Greek Capital Letter Kappa       κ   Greek Small Letter Kappa
   // Λ   Greek Capital Letter Lambda       λ   Greek Small Letter Lambda
   // Μ  Greek Capital Letter Mu       μ   Greek Small Letter Mu
   // Ν  Greek Capital Letter Nu        ν   Greek Small Letter Nu
   // Ξ   Greek Capital Letter Xi         ξ   Greek Small Letter Xi
   // Ο  Greek Capital Letter Omicron      ο   Greek Small Letter Omicron
   // Π  Greek Capital Letter Pi          π   Greek Small Letter Pi
   // Ρ   Greek Capital Letter Rho      ρ   Greek Small Letter Rho
   // Σ   Greek Capital Letter Sigma       ς   Greek Small Letter Final Sigma
   //                       σ   Greek Small Letter Sigma
   // Τ   Greek Capital Letter Tau         τ   Greek Small Letter Tau
   // Υ   Greek Capital Letter Upsilon     υ   Greek Small Letter Upsilon
   // Φ  Greek Capital Letter Phi       φ  Greek Small Letter Phi
   // Χ   Greek Capital Letter Chi       χ   Greek Small Letter Chi
   // Ψ  Greek Capital Letter Psi        ψ  Greek Small Letter Psi
   // 
   // 
   // 
   // ▄▄▄▄▄▄▄▄▄▄▄▄▄▄▄▄▄▄▄▄▄▄▄▄▄▄▄▄▄▄▄▄▄▄▄▄▄▄▄▄▄▄▄▄
   // INDEXING CHARACTERS  (all characters are 1 EM wide)
   // 
   // 
   // ① Circled One              ⑴ Bracketed One           ⒈ One Full Stop
   // ② Circled Two              ⑵ Bracketed Two           ⒉ Two Full Stop
   // ③ Circled Three              ⑶ Bracketed Three           ⒊ Three Full Stop
   // ④ Circled Four             ⑷ Bracketed Four             ⒋ Four Full Stop
   // ⑤ Circled Five              ⑸ Bracketed Five           ⒌ Five Full Stop
   // ⑥ Circled Six             ⑹ Bracketed Six             ⒍ Six Full Stop
   // ⑦ Circled Seven             ⑺ Bracketed Seven          ⒎ Seven Full Stop
   // ⑧ Circled Eight            ⑻ Bracketed Eight            ⒏ Eight Full Stop
   // ⑨ Circled Nine             ⑼ Bracketed Nine          ⒐ Nine Full Stop
   // ⑩ Circled Ten            ⑽ Bracketed Ten            ⒑ Ten Full Stop
   // ⑪ Circled Eleven            ⑾ Bracketed Eleven         ⒒ Eleven Full Stop
   // ⑫ Circled Twelve            ⑿ Bracketed Twelve         ⒓ Twelve Full Stop
   // ⑬ Circled Thirteen             ⒀ Bracketed Thirteen          ⒔ Thirteen Full Stop
   // ⑭ Circled Fourteen           ⒁ Bracketed Fourteen        ⒕ Fourteen Full Stop
   // ⑮ Circled Fifteen            ⒂ Bracketed Fifteen         ⒖ Fifteen Full Stop
   // ⑯ Circled Sixteen           ⒃ Bracketed Sixteen           ⒗ Sixteen Full Stop
   // ⑰ Circled Seventeen           ⒄ Bracketed Seventeen        ⒘ Seventeen Full Stop
   // ⑱ Circled Eighteen           ⒅ Bracketed Eighteen        ⒙ Eighteen Full Stop
   // ⑲ Circled Nineteen           ⒆ Bracketed Nineteen           ⒚ Nineteen Full Stop
   // ⑳ Circled Twenty            ⒇ Bracketed Twenty         ⒛ Twenty Full Stop
   // 
   // 
   // 
   // ▄▄▄▄▄▄▄▄▄▄▄▄▄▄▄▄▄▄▄▄▄▄▄▄▄▄▄▄▄▄▄▄▄▄▄▄▄▄▄▄▄▄▄▄
   // ROMAN NUMERALS
   // 
   // 
   // Ⅰ    Roman num One          ⅰ    Small Roman num One
   // Ⅱ   Roman num Two           ⅱ   Small Roman num Two
   // Ⅲ  Roman num Three           ⅲ  Small Roman num Three
   // Ⅳ  Roman num Four          ⅳ  Small Roman num Four
   // Ⅴ   Roman num Five          ⅴ   Small Roman num Five
   // Ⅵ  Roman num Six             ⅵ  Small Roman num Six
   // Ⅶ Roman num Seven         ⅶ    Small Roman num Seven
   // Ⅷ    Roman num Eight           ⅷ   Small Roman num Eight
   // Ⅸ  Roman num Nine            ⅸ  Small Roman num Nine
   // Ⅹ   Roman num Ten           ⅹ   Small Roman num Ten
   // Ⅺ  Roman num Eleven           ⅺ  Small Roman num Eleven
   // Ⅻ Roman num Twelve           ⅻ  Small Roman num Twelve
   // Ⅼ   Roman num Fifty           ⅼ    Small Roman num Fifty
   // Ⅽ   Roman num One Hundred        ⅽ   Small Roman num One Hundred
   // Ⅾ  Roman num Five Hundred      ⅾ   Small Roman num Five Hundred
   // Ⅿ  Roman num One Thousand      ⅿ     Small Roman num One Thousand    
   // 
   // 
   // ████████████████████ END    ████████████████████
END_REGION

REGION Network 16: Special characters — Mathematical operators (including vulgar fractions)
   // ▄▄▄▄▄▄▄▄▄▄▄▄▄▄▄▄▄▄▄▄▄▄▄▄▄▄▄▄▄▄▄▄▄▄▄▄▄▄▄▄▄▄▄▄
   // MATHEMATICAL OPERATORS
   // 
   // 
   // ×   Multiplication Sign          ¹   Superscript One           ∅  Empty Set
   // ÷   Division Sign              ²   Superscript Two            ∈  Element Of
   // +   Plus sign                ³   Superscript Three         ∉  Not An Element Of
   // −   Minus Sign            ½  Vulgar Fraction One Half         ∊   Small Element Of
   // ⁒   Commercial Minus Sign       ⅓  Vulgar Fraction One Third       ∋  Contains As Member
   // ±   Plus-Minus Sign             ⅔  Vulgar Fraction Two Thirds      ∌  Does Not Contain As Member
   // ∓   Minus-Or-Plus Sign          ¼  Vulgar Fraction One Quarter        ∍   Small Contains As Member
   // ≤   Less-Than Or Equal To       ¾  Vulgar Fraction Three Quarters      ∩   Intersection
   // ≥   Greater-Than Or Equal To        ⅕  Vulgar Fraction One Fifth        ∪   Union
   // ≪  Much Less-Than            ⅖  Vulgar Fraction Two Fifths       ⊂  Subset Of
   // ≫  Much Greater-Than          ⅗  Vulgar Fraction Three Fifths       ⊃  Superset Of
   // √  Square Root             ⅘  Vulgar Fraction Four Fifths      ⊄  Not A Subset Of
   // ∛  Cube Root             ⅙  Vulgar Fraction One Sixth       ⊅  Not A Superset Of
   // ∜  Fourth Root              ⅚  Vulgar Fraction Five Sixths        ⊆  Subset Of Or Equal To
   // ∝  Proportional To           ⅛  Vulgar Fraction One Eighth       ⊇  Superset Of Or Equal To
   // ∞  Infinity              ⅜  Vulgar Fraction Three Eighths      ⊈  not A Subset Of Nor Equal To
   // °   Degree Sign            ⅝  Vulgar Fraction Five Eighths     ⊉  not A Superset Of Nor Equal To
   // µ   Micro Sign             ⅞  Vulgar Fraction Seven Eighths    ⊊  Subset Of Not Equal To
   // ‰   Per Mille Sign              ⅟   Fraction Numerator One         ⊋  Superset Of Not Equal To
   // ‱  Per Ten Thousand& Sign          ⁄    Fraction Slash            ⊌   Multiset
   // ∀  For All                                    ⊍   Multiset Multiplication
   // ∁   Complement                                 ⊎   Multiset Union
   // ∂   Partial Differential                              ⊏  Square Image Of
   // ∃   There Exists                                ⊐  Square Original Of
   // ∄   There Does Not Exist          ∆   Increment             ⊑  Square Image Of Or Equal To
   // ∴    Therefore               ∇  Nabla               ⊒  Square Original Of Or Equal To
   // ∵    Because                                   ⊓  Square Cap
   // ∶   Ratio                                   ⊔  Square Cup
   // ∷  Proportion    
   // ∿  Sine Wave    
   //      
   // ∥   Parallel To             ∫    Integral               ⌠    Top Half Integral
   // ∦   Not Parallel To            ∬    Dbl Integral              ⌡    Bottom Half Integral
   // ∟ Right Angle              ∭   Triple Integral             ❲   Light Left Shell Bracket 
   // ⊾  Right Angle Arc           ∮   Contour Integral           ❳   Light Right Shell Bracket 
   // ⊿  Right Triangle             ∯    Surface Integral            ⟪   Maths Left dbl Angle Bracket
   // ∠  Angle               ∰   Volume Integral            ⟫   Maths Right dbl Angle Bracket
   // ∡  Measured Angle           ∱   Clockwise Integral           ⟬   Maths Left White Shell Bracket
   // ∢  Spherical Angle            ∲   Clockwise Contour Integral       ⟭   Maths Right White Shell Bracket
   // ⌒    Arc                 ∳   Anticlockwise Contour Integral
   // ⌓    Segment    
   // ⌔     Sector    
   // 
   // ≃   Asymptotically Equal To       ⊕    Circled Plus              ′    Prime
   // ≄   Not Asymptotically Equal To      ⊖    Circled Minus              ″    Dbl Prime
   // ≅   Approx Equal To            ⊗    Circled Times              ‴   Triple Prime
   // ≆   Approx But Not Actually Equal To    ⊘    Circled Division Slash        ⁗   Quadruple Prime
   // ≇   Not approx Nor Actually Equal To   ⊙    Circled Dot Operator          ‵    Reversed Prime
   // ≈   Almost Equal To            ⊚    Circled Ring Operator        ‶    Reversed dbl Prime
   // ≉  Not Almost Equal To          ⊛    Circled Asterisk Operator        ‷   Reversed Triple Prime
   // ≊   Almost Equal Or Equal To       ⊜    Circled Equals
   // ≋   Triple Tilde             ⊝    Circled Dash
   // ≌   All Equal To              ⊞    Squared Plus
   // ≍  Equivalent To             ⊟    Squared Minus
   // ≡   Identical To              ⊠    Squared Times
   // ≢   Not Identical To             ⊡    Squared Dot Operator
   //      
   // ∧  Logical &               ⊢  Right Tack              °   Degree Sign
   // ∨  Logical Or             ⊣  Left Tack                ℃    Degree Celsius
   // ⊻  Xor                 ⊤  Down Tack               ℉    Degree Fahrenheit
   // ⊼  Nand                ⊥  Up Tack                Ω    Ohm Sign    
   // 
   // 
   // ██████████████ █ █ █ █  END   █ █ █ █ ██████████████
END_REGION

